(*******************************************************************)
(* Trigger  *)
(*******************************************************************)
(* Zurücksetzen *)
IF xIN_RESET THEN
    iPreStep  := ST160_CETA_e.RESET;
    iOUT_Step := ST160_CETA_e.RESET;
END_IF;

(* Error Quittieren *)
IF (bOUT_Error <> 0) AND xIN_Quit THEN
    xOUT_ErrFlag := FALSE;
    bOUT_Error   := 0;
    iOUT_Step    := ST160_CETA_e.INIT;
END_IF;

(*******************************************************************)
(* Timer *)
(*******************************************************************)
TON_Timeout(IN := xIN_NextStep AND (iLastStep = iOUT_Step) (*todo FG *) ,
            PT := tIN_Timeout);

(*******************************************************************)
(* Bausteine *)
(*******************************************************************)
fb_PnpVerAxis(config          := axis_01Z_LinearConfig,
              xIN_Init        := enIN_State = enState.StateINIT,
              xIN_Reset       := xIN_Reset,
              lrIN_CurrPos    := fb_axis160_01Z.rOUT_ActPos,
              lrIN_Delta_mm   := 0.05,
              iIN_CurrentStep := iOUT_Step,
              iIN_moveNumber  := ST160_PnpVerPos_e._max);

simu_axis160_01Z(xIN_InSimu    := CETA_SIMULATION AND CONST.USE_SIMULATION,
                 rIN_PosActual := fb_axis160_01Z.rOUT_ActPos,
                 pIN_axisSimu  := ADR(axisRef_Simulation),
                 pIN_axisHW    := ADR(axisRef_Hardware),
                 rIN_PosMax    := constAxis_01Z_Beckhoff.POS_MAX,
                 rIN_PosMin    := constAxis_01Z_Beckhoff.POS_MIN,
                 rIN_PixMax    := 80,
                 rIN_PixMin    := 0);

fb_axis160_01Z(enIN_State       := enIN_State,
               parIN_Buttons    := axis_01Z_parIN_Buttons,
               xIN_DisButtons   :=,
               xIN_Quit         := xIN_Quit,
               xIN_AX5000       := TRUE,
               xIN_ENC_ABS      := TRUE, // TODO set accordingly
               xIN_PARAMok      := TRUE,
               xIN_FREE         := TRUE,
               xIN_FREE_HOME    := TRUE,
               rIN_POSMIN       := constAxis_01Z_Beckhoff.POS_MIN,
               rIN_POSMAX       := constAxis_01Z_Beckhoff.POS_MAX,
               rIN_VELOMAX      := constAxis_01Z_Beckhoff.VELO_MAX,
               rIN_VELOMANU     := constAxis_01Z_Beckhoff.VELO_MANU,
               rIN_VELOOPEN     := constAxis_01Z_Beckhoff.POS_MAX / 4,
               rIN_JogInc       := AXIS.rTeachIncAxis,
               rIN_VeloJogManu  := TO_REAL(AXIS.rJogVelo_pc),
               xIN_HomeExe      :=,
               xIN_HomeCalib    :=,
               xIN_Execute      := fb_PnpVerAxis.xOUT_Execute,
               xIN_HomeExe      :=,
               xIN_Relative     :=,
               rIN_Position     := TO_REAL(fb_PnpVerAxis.OUT_MoveProfile.lrPosition),
               rIN_Velocity     := TO_REAL(fb_PnpVerAxis.OUT_MoveProfile.lrVelocity),
               rIN_Acceleration := TO_REAL(fb_PnpVerAxis.OUT_MoveProfile.lrAccel),
               rIN_Deceleration := TO_REAL(fb_PnpVerAxis.OUT_MoveProfile.lrDecel),
               rIN_Jerk         := TO_REAL(fb_PnpVerAxis.OUT_MoveProfile.lrJerk),
               rIN_PosManu      := TO_REAL(axis_01Z_LinearConfig
                                               .movesList[AXIS.bTeachPos[iSelectedAxis]].lrPosition),
               xIN_Reset := (ST160_CETA_e.RESET = iOUT_Step) OR xIN_Reset,
               // output
               rOUT_ActPos => refAxis_01Z_beckhoff.rActPos,
               axisIN_REF  := simu_axis160_01Z.pOUT_axisRef^);

// pneumatics
fb_capMainteningLeft(xIN_Reset    := xIN_Reset OR (ST160_CETA_e.RESET = iOUT_Step),
                     xIN_Quit     := xIN_Quit,
                     xIN_Manu     := enState.StateMANU = enIN_State,
                     pbtIN_Button := ADR(refCylinderBp[1]),
                     xIN_GS       := simu_capMainteningLeft.xOUT_inGS,
                     xIN_AS       := simu_capMainteningLeft.xOUT_inAS,
                     xIN_FREE     := TRUE,
                     xINtoGS      := (ST160_CETA_e.Init_pneumatics = iOUT_Step) OR
                                     (ST160_CETA_e.handling_up = iOUT_Step),
                     xINtoAS   := IN_recipe.Use_element_left AND (ST160_CETA_e.handling_down = iOUT_Step),
                     tIN_ErrAS := DINT_TO_TIME(refCylinderConf
                                                   [ST160_Cylinders_e.Niederhalter_links].toAS_alarm_time),
                     tIN_ErrGS := DINT_TO_TIME(refCylinderConf
                                                   [ST160_Cylinders_e.Niederhalter_links].toGS_alarm_time),
                     tIN_WaitAS := DINT_TO_TIME(refCylinderConf
                                                    [ST160_Cylinders_e.Niederhalter_links].toAS_wait_time),
                     tIN_WaitGS := DINT_TO_TIME(refCylinderConf
                                                    [ST160_Cylinders_e.Niederhalter_links].toGS_wait_time));

simu_capMainteningLeft(xIN_Enable := TRUE, // CETA_SIMULATION AND CONST.USE_SIMULATION,
                       xIN_inGS   := UINT_TO_INT(uiIN_DisplacementSensorLeft) < 10,
                       xIN_inAS   := UINT_TO_INT(uiIN_DisplacementSensorLeft) > 200,
                       xIN_valve  := fb_capMainteningLeft.xOUT_VALVE,
                       tIN_GS_ms  := 200,  // ms
                       tIN_AS_ms  := 200); // ms

fb_capMainteningRight(xIN_Reset    := xIN_Reset OR (ST160_CETA_e.RESET = iOUT_Step),
                      xIN_Quit     := xIN_Quit,
                      xIN_Manu     := enState.StateMANU = enIN_State,
                      pbtIN_Button := ADR(refCylinderBp[2]),
                      xIN_GS       := simu_capMainteningRight.xOUT_inGS,
                      xIN_AS       := simu_capMainteningRight.xOUT_inAS,
                      xIN_FREE     := TRUE,
                      xINtoGS      := (ST160_CETA_e.Init_pneumatics = iOUT_Step) OR
                                      (ST160_CETA_e.handling_up = iOUT_Step),
                      xINtoAS := IN_recipe.Use_element_right AND (ST160_CETA_e.handling_down = iOUT_Step),
                      tIN_ErrAS
                          := DINT_TO_TIME(refCylinderConf
                                              [ST160_Cylinders_e.Niederhalter_rechts].toAS_alarm_time),
                      tIN_ErrGS := DINT_TO_TIME(refCylinderConf
                                                    [ST160_Cylinders_e.Niederhalter_rechts].toGS_alarm_time),
                      tIN_WaitAS := DINT_TO_TIME(refCylinderConf
                                                     [ST160_Cylinders_e.Niederhalter_rechts].toAS_wait_time),
                      tIN_WaitGS := DINT_TO_TIME(refCylinderConf
                                                     [ST160_Cylinders_e.Niederhalter_rechts].toGS_wait_time));

simu_capMainteningRight(xIN_Enable := TRUE, // CETA_SIMULATION AND CONST.USE_SIMULATION,
                        xIN_inGS   := UINT_TO_INT(uiIN_DisplacementSensorRight) < 10,
                        xIN_inAS   := UINT_TO_INT(uiIN_DisplacementSensorRight) > 200,
                        xIN_valve  := fb_capMainteningRight.xOUT_VALVE,
                        tIN_GS_ms  := 200,  // ms
                        tIN_AS_ms  := 200); // ms

fb_dichtung_left(xIN_Reset    := xIN_Reset OR (ST160_CETA_e.RESET = iOUT_Step),
                 xIN_Quit     := xIN_Quit,
                 xIN_Manu     := enState.StateMANU = enIN_State,
                 pbtIN_Button := ADR(refCylinderBp[3]),
                 xIN_GS       := simu_dichtung_left.xOUT_inGS,
                 xIN_AS       := simu_dichtung_left.xOUT_inAS,
                 xIN_FREE     := TRUE,
                 xINtoGS      := (ST160_CETA_e.Init_pneumatics = iOUT_Step) OR
                                 (ST160_CETA_e.unseal_piece = iOUT_Step),
                 xINtoAS   := IN_recipe.Use_element_left AND (ST160_CETA_e.seal_piece = iOUT_Step),
                 tIN_ErrAS := DINT_TO_TIME(refCylinderConf
                                               [ST160_Cylinders_e.Dichtung_prufglocke_links].toAS_alarm_time),
                 tIN_ErrGS := DINT_TO_TIME(refCylinderConf
                                               [ST160_Cylinders_e.Dichtung_prufglocke_links].toGS_alarm_time),
                 tIN_WaitAS := DINT_TO_TIME(refCylinderConf
                                                [ST160_Cylinders_e.Dichtung_prufglocke_links].toAS_wait_time),
                 tIN_WaitGS := DINT_TO_TIME(refCylinderConf
                                                [ST160_Cylinders_e.Dichtung_prufglocke_links].toGS_wait_time));

simu_dichtung_left(xIN_Enable := TRUE,                             // CETA_SIMULATION AND CONST.USE_SIMULATION,
                   xIN_inGS   := NOT fb_dichtung_right.xOUT_VALVE, // no sensor here
                   xIN_inAS   := fb_dichtung_right.xOUT_VALVE,     // no sensor here
                   xIN_valve  := fb_dichtung_left.xOUT_VALVE,
                   tIN_GS_ms  := 200,  // ms
                   tIN_AS_ms  := 200); // ms

fb_dichtung_right(xIN_Reset    := xIN_Reset OR (ST160_CETA_e.RESET = iOUT_Step),
                  xIN_Quit     := xIN_Quit,
                  xIN_Manu     := enState.StateMANU = enIN_State,
                  pbtIN_Button := ADR(refCylinderBp[4]),
                  xIN_GS       := simu_dichtung_right.xOUT_inGS,
                  xIN_AS       := simu_dichtung_right.xOUT_inAS,
                  xIN_FREE     := TRUE,
                  xINtoGS      := (ST160_CETA_e.Init_pneumatics = iOUT_Step) OR
                                  (ST160_CETA_e.unseal_piece = iOUT_Step),
                  xINtoAS   := IN_recipe.Use_element_right AND (ST160_CETA_e.seal_piece = iOUT_Step),
                  tIN_ErrAS := DINT_TO_TIME(refCylinderConf
                                                [ST160_Cylinders_e.Dichtung_prufglocke_rechts].toAS_alarm_time),
                  tIN_ErrGS := DINT_TO_TIME(refCylinderConf
                                                [ST160_Cylinders_e.Dichtung_prufglocke_rechts].toGS_alarm_time),
                  tIN_WaitAS := DINT_TO_TIME(refCylinderConf
                                                 [ST160_Cylinders_e.Dichtung_prufglocke_rechts].toAS_wait_time),
                  tIN_WaitGS := DINT_TO_TIME(refCylinderConf
                                                 [ST160_Cylinders_e.Dichtung_prufglocke_rechts].toGS_wait_time));

simu_dichtung_right(xIN_Enable := TRUE,                             // CETA_SIMULATION AND CONST.USE_SIMULATION,
                    xIN_inGS   := NOT fb_dichtung_right.xOUT_VALVE, // no sensor here
                    xIN_inAS   := fb_dichtung_right.xOUT_VALVE,     // no sensor here
                    xIN_valve  := fb_dichtung_right.xOUT_VALVE,
                    tIN_GS_ms  := 200,  // ms
                    tIN_AS_ms  := 200); // ms

(*******************************************************************)
(* OUTPUTS *)
(*******************************************************************)
// Error Flag 
xOUT_ErrFlag := (bOUT_Error <> 0) OR (ST160_CETA_e.ERROR = iOUT_Step);
// Baustein befindet sich im Ablauf 
xOUT_Busy := (iOUT_Step > ST160_CETA_e.READY) AND (iOUT_Step < ST160_CETA_e.DONE);
// Baustein hat den Ablauf beendet
xOUT_Done := (iOUT_Step = ST160_CETA_e.DONE);
// Process ready
xOUT_Ready := (iOUT_Step = ST160_CETA_e.READY) OR (iOUT_Step = ST160_CETA_e.waitOnMover);
// Timeout FB 				 		
xOUT_Timeout := TON_Timeout.Q;
// Itialisierung fertig			
xOUT_InitDone := (iOUT_Step = ST160_CETA_e.READY) OR (iOUT_Step = ST160_CETA_e.waitOnMover);
// Aktueller Schritt			
iOUT_Step := iOUT_Step; //Im Ablauf gesetzt		
sOUT_Step := TO_STRING(iOUT_Step);
//Fehlernummer	 
bOUT_Error := bOUT_Error; //Im Ablauf/FB gesetzt	
(* Warte (alle Schritte wo auf FG oder Teile gewartet wird) *)
xOUT_Wait := (iOUT_Step = ST160_CETA_e.DONE) OR
             (iOUT_Step = ST160_CETA_e.READY) OR
             (iOUT_Step = ST160_CETA_e.START) OR
             (iOUT_Step = ST160_CETA_e.waitOnMover) OR
             (iOUT_Step = ST160_CETA_e.SYNC_MOVER_LEAVE);

xOUT_MoverFree :=
    NOT (iOUT_Step >= ST160_CETA_e.MOVER_NEEDED_OP AND iOUT_Step < ST160_CETA_e.MOVER_FREE_OP) AND
    (iOUT_Step >= ST160_CETA_e.READY) AND
    (iOUT_Step < ST160_CETA_e.ERROR);

iOUT_ProcessCompletion := F_GetPercent_2(iAktStep,
                                         iAktStep,
                                         iAktStep,
                                         ST160_CETA_e.Init_pneumatics,
                                         ST160_CETA_e.SYNC_MOVER_LEAVE);

xOUT_niederhalter_links :=
    fb_capMainteningLeft.xOUT_VALVE AND NOT (CETA_SIMULATION AND CONST.USE_SIMULATION);

xOUT_niederhalter_rechts :=
    fb_capMainteningRight.xOUT_VALVE AND NOT (CETA_SIMULATION AND CONST.USE_SIMULATION);

xOUT_dichtung_pruflocker_links :=
    fb_dichtung_left.xOUT_VALVE AND NOT (CETA_SIMULATION AND CONST.USE_SIMULATION);

xOUT_dichtung_pruflocker_rechts :=
    fb_dichtung_right.xOUT_VALVE AND NOT (CETA_SIMULATION AND CONST.USE_SIMULATION);

(*******************************************************************)
(* Ablauf *)
(*******************************************************************)

(* Sperren *)
IF xIN_Sperre THEN
    iPreStep  := ST160_CETA_e.RESET;
    iOUT_Step := ST160_CETA_e.RESET;
    RETURN;
END_IF;

(* Schritt Merker *)
IF iAktStep <> iOUT_Step THEN
    iLastStep := iAktStep;
    iAktStep  := iOUT_Step;
END_IF

(* START *)
rtSTART(CLK := xIN_Start);

IF 0 = bOUT_Error THEN
    IF fb_axis160_01Z.xOUT_ErrFlag THEN
        bOUT_Error := 11;
    ELSIF fb_capMainteningLeft.xOUT_ErrFlag THEN
        bOUT_Error := 12;
    ELSIF fb_capMainteningRight.xOUT_ErrFlag THEN
        bOUT_Error := 13;
    END_IF
ELSIF iOUT_Step < ST160_CETA_e.ERROR THEN
    iOUT_Step := ST160_CETA_e.ERROR;
END_IF

(*******************************************************************)
(* Schrittkette  *)
(*******************************************************************)
CASE iOUT_Step OF

(***** RESET *****)
ST160_CETA_e.RESET: (* Schritt 0-99 *)
    //Initialisierungen
    //Start Init Ablauf
    IF xIN_Init THEN
        iOUT_Step := ST160_CETA_e.INIT;
        //Start Manu Ablauf
    ELSIF enIN_State = StateMANU AND xIN_NextStep THEN
        iOUT_Step := ST160_CETA_e.INIT;
    END_IF;

(***** INIT *****)
ST160_CETA_e.INIT: (* Grundstellung ? *)
    iOUT_Step := ST160_CETA_e.Init_pneumatics;

ST160_CETA_e.Init_pneumatics:
    IF (fb_capMainteningLeft.xOUT_inGS AND fb_capMainteningRight.xOUT_inGS) AND
       (fb_dichtung_left.xOUT_inGS AND fb_dichtung_right.xOUT_inGS) THEN
        iOUT_Step := ST160_CETA_e.Init_vertical_down;
    END_IF

ST160_CETA_e.Init_vertical_down:
    IF fb_PnpVerAxis.MoveTo(ST160_PnpVerPos_e.gs_down).xOUT_InPos THEN
        iOUT_Step := ST160_CETA_e.Init_set_program_number;
    END_IF

ST160_CETA_e.Init_set_program_number:
    IF ref_fb_CETA.SetProgramNumber(IN_recipe.Program_number) THEN
        iOUT_Step := ST160_CETA_e.READY;
    END_IF

(***** READY / INIT DONE *****)
ST160_CETA_e.READY:   (* Start AUTO,END,LEER,STEP *)
    IF xIN_Start THEN //IF rtSTART.Q THEN
        iOUT_Step := ST160_CETA_e.START;
    END_IF

(***** START  ZYKLISCH *****)
ST160_CETA_e.START: (*  *)
    IF xIN_NextStep AND pxFG_Freigabe^ THEN
        iOUT_Step       := ST160_CETA_e.waitOnMover;
        xCETA_Result_OK := FALSE;
    END_IF;

ST160_CETA_e.waitOnMover: (*  *)
    IF xIN_NextStep AND __ISVALIDREF(Mover) THEN
        IF (Mover.GetLastStationDone() >= iIN_StationNumber) OR Mover.IsPieceBad() THEN
            iOUT_Step := ST160_CETA_e.SYNC_MOVER_LEAVE;
        ELSIF Mover.GetLastStationDone() < INT#150 THEN
            iOUT_Step := ST160_CETA_e.SYNC_MOVER_LEAVE;
        ELSE
            iOUT_Step := ST160_CETA_e.handling_down;
        END_IF
    END_IF;

ST160_CETA_e.handling_down:
    IF (NOT IN_recipe.Use_element_left OR fb_capMainteningLeft.xOUT_inAS) AND
       (NOT IN_recipe.Use_element_right OR fb_capMainteningRight.xOUT_inAS) THEN
        iOUT_Step := ST160_CETA_e.vertical_up;
    END_IF

ST160_CETA_e.vertical_up:
    IF fb_PnpVerAxis.MoveTo(ST160_PnpVerPos_e.as_up).xOUT_InPos THEN
        iOUT_Step := ST160_CETA_e.seal_piece;
    END_IF

ST160_CETA_e.seal_piece:
    IF (NOT IN_recipe.Use_element_left OR fb_dichtung_left.xOUT_inAS) AND
       (NOT IN_recipe.Use_element_right OR fb_dichtung_right.xOUT_inAS) THEN
        IF CETA_SIMULATION AND CONST.USE_SIMULATION THEN
            iOUT_Step       := ST160_CETA_e.unseal_piece;
            xCETA_Result_OK := TRUE;
        ELSE
            iOUT_Step := ST160_CETA_e.CETA_start;
        END_IF
    END_IF

ST160_CETA_e.CETA_start:
    IF ref_fb_CETA.xOUT_ReadyToStart THEN
        IF ref_fb_CETA.StartMeasurement() THEN
            iOUT_Step := ST160_CETA_e.CETA_wait_on_result;
        ELSE
            bOUT_Error := 21;
        END_IF
    END_IF

ST160_CETA_e.CETA_wait_on_result:
    IF ref_fb_CETA.xOUT_DataReady THEN
        // this void call is needed to tell CETA function block
        // that we have read the result
        ref_fb_CETA.GetResult();
        xCETA_Result_OK := ref_fb_CETA.xOUT_MeasureOK;
        iOUT_Step       := ST160_CETA_e.unseal_piece;
    END_IF

ST160_CETA_e.unseal_piece:
    IF (NOT IN_recipe.Use_element_left OR fb_dichtung_left.xOUT_inGS) AND
       (NOT IN_recipe.Use_element_right OR fb_dichtung_right.xOUT_inGS) THEN
        iOUT_Step := ST160_CETA_e.vertical_down;
    END_IF

ST160_CETA_e.vertical_down:
    IF fb_PnpVerAxis.MoveTo(ST160_PnpVerPos_e.gs_down).xOUT_InPos THEN
        iOUT_Step := ST160_CETA_e.handling_up;
    END_IF

ST160_CETA_e.handling_up:
    IF fb_capMainteningLeft.xOUT_inGS AND fb_capMainteningRight.xOUT_inGS THEN
        iOUT_Step := ST160_CETA_e.SYNC_MOVER_LEAVE;

        IF __ISVALIDREF(Mover) AND NOT xCETA_Result_OK THEN
            Mover.SetErrorCode(CONCAT(INT_TO_STRING(iIN_StationNumber), '-C'));
            // bOUT_Error := 8; // TODO Remove
            iPreStep   := ST160_CETA_e.SYNC_MOVER_LEAVE;

            IF NOT Mover.SetLastStation(-iIN_StationNumber) THEN
                ASSERT(0);
            END_IF
        ELSIF __ISVALIDREF(Mover) AND xCETA_Result_OK THEN
            IF NOT Mover.SetLastStation(iIN_StationNumber) THEN
                ASSERT(0);
            END_IF
        END_IF
    END_IF

ST160_CETA_e.SYNC_MOVER_LEAVE:
    // The mover needs to be taken by MoverMan
    IF NOT __ISVALIDREF(Mover) THEN
        iOUT_Step := ST160_CETA_e.DONE;
    END_IF

(***** DONE *****)
ST160_CETA_e.DONE: (* Letzter Schritt  *)
    IF NOT xIN_AlarmAktiv THEN
        //AUTO
        IF (enIN_State = StateAUTO) AND xIN_RestartCYCL THEN
            iOUT_Step := ST160_CETA_e.START;
            //STEP / END / LEERFAHREN restart
        ELSIF (enIN_State < StateAUTO) AND (enIN_State >= enState.StateSTEP) AND xIN_RestartCYCL THEN
            iOUT_Step := ST160_CETA_e.START;
            //STEP / END / LEERFAHREN fertig
        ELSIF (enIN_State = StateREADY) THEN
            iOUT_Step := ST160_CETA_e.READY;
        END_IF;
    END_IF;

(************ ERROR *************)
ST160_CETA_e.ERROR: (* ERROR *) ;

END_CASE;

END_FUNCTION_BLOCK

// ---- POUs/20_AUTO/ST16x/CETA/FB_CETA_715.TcPOU
// Manage CETATEST void test
// Use the method to perform actions
// Please call each method only once (Use the command only during transition between step) 
FUNCTION_BLOCK PUBLIC FB_CETA_715
VAR_INPUT
    xIN_StatusBits : CETA_IN_u;            // connect this to the 2 first byte of the input of the CETATEST
    xIN_Data       : ARRAY[0..61] OF BYTE; // connect those 62 bytes right after xIN_StatusBits
    xIN_Reset      : BOOL;                 // Reset errors
END_VAR
VAR_OUTPUT
    xOUT_CommandBits    : CETA_OUT_u;           // connect this to the 2 first byte of the Output of the CETATEST
    xOUT_Data           : ARRAY[0..29] OF BYTE; // connect those 30 bytes right after xIN_StatusBits
    xOUT_DataReady      : BOOL;
    xOUT_Error_Flag     : BOOL;
    bOUT_ErrorCode      : BYTE;
    sOUT_ErrorMessage   : STRING;
    xOUT_Measure_1_GOOD : BOOL; // TRUE when the last measurement in canal 1 was GOOD
    bOUT_Error_1        : BYTE;
    xOUT_Measure_2_GOOD : BOOL; // TRUE when the last measurement in canal 2 was GOOD
    bOUT_Error_2        : BYTE;
    xOUT_ReadyToStart   : BOOL; // you can send a start signal
END_VAR
VAR
    iStep       : INT := 0;
    ton_TimeOut : TON;

    iBlockNumber : INT := 0;

    error_message : CETA_error_handling_t;

    ceta_measurement_data : CETA_Measurement_t;

    xResultGood : BOOL := FALSE;

END_VAR
VAR CONSTANT
    DEFAULT_COMMAND_BIT : UINT := 16#00;
END_VAR


ton_TimeOut(IN := 200 = iStep OR 1100 = iStep, PT := T#10S);

CASE iStep OF

0: // reset
    xOUT_CommandBits.raw := 0;

    IF xIN_StatusBits.bits.b09_communication_possible THEN
        iStep := 100;
    END_IF

100: // ready to take command
    // wait on command and read error when there is one
    IF xIN_StatusBits.bits.b08_error_bit THEN
        iStep       := 1000;
        xResultGood := FALSE;
    END_IF

200: // command is sending, wait on a answer

    IF ton_TimeOut.Q THEN
        iStep             := 1500;
        bOUT_ErrorCode    := 0;
        sOUT_ErrorMessage := 'Command timeout';

    ELSIF xOUT_CommandBits.bits.b00_start_stop THEN
        IF xIN_StatusBits.bits.b00_measurement_complete THEN
            iStep               := 240;
            iBlockNumber        := 0;
            xOUT_Measure_1_GOOD := FALSE;
            xOUT_Measure_2_GOOD := FALSE;
        END_IF

    ELSIF xOUT_CommandBits.bits.b01_send_parameters THEN
        IF xIN_StatusBits.bits.b02_parameters_available THEN
            iStep := 300;
        END_IF

    ELSIF xOUT_CommandBits.bits.b02_request_parameters THEN
        IF xIN_StatusBits.bits.b02_parameters_available THEN
            iStep := 300;
        END_IF

    ELSIF xOUT_CommandBits.bits.b03_request_error_code THEN
        IF xIN_StatusBits.bits.b03_error_code_available THEN
            iStep := 1200;
        END_IF

    ELSIF xOUT_CommandBits.bits.b04_change_front_panel_lock_state THEN
        IF xIN_StatusBits.bits.b04_front_panel_lock_state THEN // TODO
            iStep := 0;
        END_IF

    ELSIF xOUT_CommandBits.bits.b05_assign_program_number THEN
        IF xIN_StatusBits.bits.b05_program_number_assigned THEN
            iStep := 0;
        END_IF

    ELSIF xOUT_CommandBits.bits.b06_request_system_information THEN
        IF xIN_StatusBits.bits.b06_system_information_available THEN
            iStep := 300;
        END_IF

    ELSIF xOUT_CommandBits.bits.b07_request_cycle_counter THEN
        IF xIN_StatusBits.bits.b07_cycle_counter_available THEN
            iStep := 300;
        END_IF

        // ELSIF xOUT_CommandBits.bits.request_next_result_block THEN
        //     IF xIN_StatusBits.bits.ne THEN
        //         iStep := 300;
        //     END_IF
    END_IF

240:

    iStep := 250;

    // copy 
    CASE iBlockNumber OF
    0:
        MEMCPY(ADR(ceta_measurement_data.Block0), ADR(xIN_Data), SIZEOF(ceta_measurement_data.Block0));
    1:
        MEMCPY(ADR(ceta_measurement_data.Block1), ADR(xIN_Data), SIZEOF(ceta_measurement_data.Block1));
    2:
        MEMCPY(ADR(ceta_measurement_data.Block2), ADR(xIN_Data), SIZEOF(ceta_measurement_data.Block2));

    ELSE
        iStep := 1500; // should not read more than 3 blocks !
    END_CASE

    iBlockNumber := iBlockNumber + 1;

250:

    // Here we test for iBlockNumber 1 but we have increment the value before
    IF 2 = iBlockNumber THEN
        xOUT_Measure_1_GOOD := ceta_measurement_data.Block1.Result_chanel_1 = CETA_REsult_e.OK;
        xOUT_Measure_2_GOOD := ceta_measurement_data.Block1.Result_chanel_2 = CETA_REsult_e.OK;

        IF NOT xOUT_Measure_1_GOOD THEN
            bOUT_Error_1 := ceta_measurement_data.Block1.Result_chanel_1;
        ELSE
            bOUT_Error_1 := 0;
        END_IF

        IF NOT xOUT_Measure_2_GOOD THEN
            bOUT_Error_2 := ceta_measurement_data.Block1.Result_chanel_2;
        ELSE
            bOUT_Error_2 := 0;
        END_IF
    END_IF

    IF xIN_StatusBits.bits.b11_result_block_handshake_bit THEN
        iStep := 260;
    ELSE
        iStep := 300;
    END_IF

260:
    IF NOT xIN_StatusBits.bits.b11_result_block_handshake_bit THEN
        iStep := 240;
    END_IF

    xOUT_CommandBits.bits.b11_request_next_result_block := xIN_StatusBits.bits.b11_result_block_handshake_bit;

300: // data available
    xOUT_CommandBits.raw := 0;
// Use the read() method to return to state 100

1000: // read error code
    xOUT_CommandBits.raw := 0;
    //
    xOUT_CommandBits.bits.b03_request_error_code := TRUE;

    iStep := 1100;

1100: // read error code
    IF ton_TimeOut.Q THEN
        iStep := 0; // reset .. there is nothing we can do
    ELSIF xIN_StatusBits.bits.b03_error_code_available THEN
        iStep := 1200;
    END_IF

1200: // read error
    error_message.command_in_error.raw := xIN_Data[0] + SHL(TO_UINT(xIN_Data[1]), 8);

    bOUT_ErrorCode := error_message.error_code;

    IF 0 = error_message.command_in_error.raw THEN
        sOUT_ErrorMessage := 'CETA in error, not due to Ethercat communication';

    ELSIF xOUT_CommandBits.bits.b01_send_parameters THEN
        sOUT_ErrorMessage := 'send_parameters command failed';

    ELSIF xOUT_CommandBits.bits.b02_request_parameters THEN
        sOUT_ErrorMessage := 'request_parameters command failed';

    ELSIF xOUT_CommandBits.bits.b03_request_error_code THEN
        sOUT_ErrorMessage := 'request_error_code command failed';

    ELSIF xOUT_CommandBits.bits.b04_change_front_panel_lock_state THEN
        sOUT_ErrorMessage := 'change_front_panel_lock_state command failed';

    ELSIF xOUT_CommandBits.bits.b05_assign_program_number THEN
        sOUT_ErrorMessage := 'assign_program_number command failed';

    ELSIF xOUT_CommandBits.bits.b06_request_system_information THEN
        sOUT_ErrorMessage := 'request_system_information command failed';

    ELSIF xOUT_CommandBits.bits.b07_request_cycle_counter THEN
        sOUT_ErrorMessage := 'request_cycle_counter command failed';

    END_IF

    iStep := 1500;

1500: // in error, wait on reset
    IF xIN_Reset THEN
        sOUT_ErrorMessage                         := '';
        bOUT_ErrorCode                            := 0;
        xOUT_CommandBits.raw                      := 0;
        xOUT_CommandBits.bits.b08_reset_error_bit := TRUE;
        iStep                                     := 0;
    END_IF

END_CASE

xOUT_DataReady    := 300 = iStep;
xOUT_Error_Flag   := 1500 = iStep;
xOUT_ReadyToStart := xIN_StatusBits.bits.b10_device_ready_to_start;

METHOD GetParameter : BOOL
VAR_INPUT
END_VAR
END_METHOD

METHOD GetResult : BOOL
VAR_INPUT
END_VAR
IF 300 = THIS^.iStep THEN
    GetResult   := TRUE;
    THIS^.iStep := 0;
ELSE
    GetResult := FALSE;
END_IF
END_METHOD

METHOD SetProgramNumber : BOOL
VAR_INPUT
	program_number : USINT;
END_VAR
IF 100 = THIS^.iStep THEN
	THIS^.iStep := 200;
	THIS^.xOUT_CommandBits.bits.b05_assign_program_number := TRUE;
	THIS^.xOUT_Data[0] := USINT_TO_BYTE(program_number);
	SetProgramNumber := TRUE;
ELSE
    THIS^.iStep      := 0;
	SetProgramNumber := FALSE;
END_IF
END_METHOD

METHOD StartMeasurement : BOOL
VAR_INPUT
END_VAR
IF 100 = THIS^.iStep THEN
    THIS^.iStep                                := 200;
    THIS^.xOUT_CommandBits.bits.b00_start_stop := TRUE;
    StartMeasurement                           := TRUE;
ELSE
    THIS^.iStep      := 0;
    StartMeasurement := FALSE;
END_IF
END_METHOD

END_FUNCTION_BLOCK

// ---- POUs/20_AUTO/ST16x/FB_AUT_165.TcPOU
FUNCTION_BLOCK FB_AUT_165 EXTENDS FB_AUT_ABSTRACT
(****************************************************************************)
(*	POU_AUT_zxx			Bausteinaufrufe Station	zxx							*)
(*	Status				ungetestet											*)
(*  Version:			1.0													*)
(*	Beschrieb:																*)
(*																			*)
(*	Abläufe:			FB_ABLzxxA		Hauptablauf							*)
(*																			*)
(*																			*)
(* 	25.09.2019/Dj															*)
(****************************************************************************)
(*	dd.mm.yyyy   KZ    x.y			Beschrieb								*)
(****************************************************************************)
VAR_INPUT
    (* spezifische Eingänge *)

END_VAR
VAR_OUTPUT
    (* spezifische Ausgänge *)

END_VAR
VAR
    (* Bausteine *)
    fb_ABL_CETA : FB_ABL_160;
	
	fb_CETA : FB_CETA_715;

    fb_stat : FB_AUT_Statistics;

END_VAR

(*******************************************************************)
(* Timer *)
(*******************************************************************)

(*******************************************************************)
(* Flanken / Merker *)
(*******************************************************************)
//MANU CYCLE
IF (enIN_State = StateMANU) AND xIN_ManuCycle THEN
    xManuCycle := TRUE;
END_IF;

IF (enIN_State <> StateMANU) OR xOUT_Done THEN
    xManuCycle := FALSE;
END_IF

//NEXT STEP
xNextStep := (enIN_State > StateSTEP) OR
             ((enIN_State = StateSTEP) AND xIN_Step) OR
             ((enIN_State = StateMANU) AND xManuCycle);

//RESET
xReset := (enIN_State < StateREADY) AND (enIN_State <> StateINIT) AND NOT xManuCycle;

(*******************************************************************)
(* Bausteinaufrufe Abläufe *)
(*******************************************************************)

xRelease := MAIN.MoverMan.IsProcessUsed(THIS^);

fb_CETA(xIN_StatusBits   := CETA_IO.I_ST165_StatusBits,
        xIN_Data         := CETA_IO.I_ST165_Data,
        xIN_Reset        := xReset OR xIN_Quit,
        xOUT_CommandBits => CETA_IO.Q_ST165_CommandBits,
        xOUT_Data        => CETA_IO.Q_ST165_Data);

fb_ABL_CETA(xIN_Reset       := xReset,
            xIN_Init        := xIN_Init,
            xIN_Quit        := xIN_Quit,
            xIN_Start       := enIN_State >= enState.StateLEER AND xRelease,
            xIN_Sperre      := NOT xIN_On,
            xIN_NextStep    := xNextStep,
            xIN_AlarmAktiv  := xIN_AlarmAktiv,
            xIN_DryCycle    := xIN_DryCycle,
            xIN_RestartCYCL := enIN_State >= enState.StateLEER,
            enIN_State      := enIN_State,
            tIN_Timeout     := tIN_Timeout,
            pxFG_Freigabe   := ADR(xRelease),
            // CleverTrackLib
            Mover := THIS^.Mover,
            // for multiple reference of the FB
            ref_fb_CETA := fb_CETA,

            refAxis_01Z_beckhoff         := ST16x_Axis.axis165_01Z,
            constAxis_01Z_Beckhoff       := ST16x_Axis.const165_01Z,
            axis_01Z_LinearConfig        := _20_AUTO.recipe.linearAxis[LinearAxis_e.ST165_01Z],
            iSelectedAxis                := Axis_e.ST165_01Z,
            axis_01Z_parIN_Buttons       := ADR(AXIS.btTeachArAxis[Axis_e.ST165_01Z]),
            refCylinderBp                := HMI.btManuCylinders[StationList_e.ST165],
            refCylinderConf              := _20_AUTO.recipe.cylinder2Pos[StationList_e.ST165],
            uiIN_DisplacementSensorLeft  := IO_BOX.I3200_ST165_Wegmessenor_links,
            uiIN_DisplacementSensorRight := IO_BOX.I3300_ST165_Wegmessenor_rechts,
            IN_recipe                    := _20_AUTO.recipe.st165,
            iIN_StationNumber            := 165,

            xOUT_niederhalter_links         => IO_BOX.Q0304_14_ST165_niederhalter_links,
            xOUT_niederhalter_rechts        => IO_BOX.Q0305_14_ST165_niederhalter_rechts,
            xOUT_dichtung_pruflocker_links  => IO_BOX.Q0306_14_ST165_dichtung_pruflocker_links,
            xOUT_dichtung_pruflocker_rechts => IO_BOX.Q0306_12_ST165_dichtung_pruflocker_rechts,

            axisRef_Hardware   := ST16x_Axis.axis165_01Z.axis,
            axisRef_Simulation := SIMU.axis_ref[Axis_e.ST165_01Z]);
			
fb_stat(xIN_Enable  := enState.StateAUTO = enIN_State,
        xIN_Waiting := fb_ABL_CETA.xOUT_Wait,
        xIN_Running := (fb_ABL_CETA.iOUT_Step >= ST160_CETA_e.START) AND
                       (fb_ABL_CETA.iOUT_Step <= ST160_CETA_e.DONE),
        // Since we use a mover system, a cycle is done when we are waiting on a mover
        xIN_Done := fb_ABL_CETA.iOUT_Step = ST160_CETA_e.waitOnMover);

(*******************************************************************)
(* Mover reset flags *)
(*******************************************************************)

(*******************************************************************)
(* OUTPUT *)
(*******************************************************************)
xOUT_InitDone := fb_ABL_CETA.xOUT_InitDone;
xOUT_Ready    := fb_ABL_CETA.xOUT_Ready;
xOUT_Done     := fb_ABL_CETA.xOUT_Done;
xOUT_ErrFlag  := fb_ABL_CETA.xOUT_ErrFlag;
xOUT_Wait     := fb_ABL_CETA.xOUT_Wait;
xOUT_AlarmST  := xOUT_ErrFlag;

(*******************************************************************)
(* Bausteinaufruf Error Station *)
(*******************************************************************)
// POU_ERR_VORLAGE(xIN_QUIT:=xIN_Quit , pstrArIN_ALARM:=ADR(HMI.strArALARM[1]));

(* % of completion of the process *)
PROPERTY iCompletionPC : INT
GET
iCompletionPC := THIS^.fb_ABL_CETA.iOUT_ProcessCompletion;
END_GET
END_PROPERTY

PROPERTY ProcessExecution : ProcessExecution_e
GET
ProcessExecution := THIS^._ProcessExecution;
END_GET
SET
THIS^._ProcessExecution := ProcessExecution;
END_SET
END_PROPERTY

PROPERTY xBusy : BOOL
GET
xBusy := THIS^.fb_ABL_CETA.xOUT_Busy;
END_GET
SET
END_SET
END_PROPERTY

PROPERTY xDone : BOOL
GET
xDone := THIS^.fb_ABL_CETA.xOUT_Ready OR THIS^.fb_ABL_CETA.xOUT_Done;
END_GET
END_PROPERTY

PROPERTY xMoverPathFree : BOOL
GET
xMoverPathFree := THIS^.fb_ABL_CETA.xOUT_MoverFree OR THIS^.fb_ABL_CETA.xOUT_Ready OR THIS^.fb_ABL_CETA.xOUT_Done;
END_GET
END_PROPERTY

PROPERTY xMoverShouldLeave : BOOL
GET
xMoverShouldLeave := THIS^.fb_ABL_CETA.iOUT_Step = ST160_CETA_e.SYNC_MOVER_LEAVE;
END_GET
END_PROPERTY

END_FUNCTION_BLOCK

// ---- POUs/20_AUTO/ST170/FB_AUT_170.TcPOU
FUNCTION_BLOCK FB_AUT_170 EXTENDS FB_AUT_ABSTRACT
(****************************************************************************)
(*	POU_AUT_zxx			Bausteinaufrufe Station	zxx							*)
(*	Status				ungetestet											*)
(*  Version:			1.0													*)
(*	Beschrieb:																*)
(*																			*)
(*	Abläufe:			FB_ABLzxxA		Hauptablauf							*)
(*																			*)
(*																			*)
(* 	25.09.2019/Dj															*)
(****************************************************************************)
(*	dd.mm.yyyy   KZ    x.y			Beschrieb								*)
(****************************************************************************)
VAR_INPUT
    (* spezifische Eingänge *)

END_VAR
VAR_OUTPUT
    (* spezifische Ausgänge *)

END_VAR
VAR
    (* Bausteine *)
    fb_ABL_RFID : FB_ABL_170;

    fb_stat : FB_AUT_Statistics;

END_VAR

(*******************************************************************)
(* Timer *)
(*******************************************************************)

(*******************************************************************)
(* Flanken / Merker *)
(*******************************************************************)
//MANU CYCLE
IF (enIN_State = StateMANU) AND xIN_ManuCycle THEN
    xManuCycle := TRUE;
END_IF;

IF (enIN_State <> StateMANU) OR xOUT_Done THEN
    xManuCycle := FALSE;
END_IF

//NEXT STEP
xNextStep := (enIN_State > StateSTEP) OR
             ((enIN_State = StateSTEP) AND xIN_Step) OR
             ((enIN_State = StateMANU) AND xManuCycle);

//RESET
xReset := (enIN_State < StateREADY) AND (enIN_State <> StateINIT) AND NOT xManuCycle;

(*******************************************************************)
(* Bausteinaufrufe Abläufe *)
(*******************************************************************)

xRelease := MAIN.MoverMan.IsProcessUsed(THIS^);

fb_ABL_RFID(xIN_Reset       := xReset,
            xIN_Init        := xIN_Init,
            xIN_Quit        := xIN_Quit,
            xIN_Start       := enIN_State >= enState.StateLEER AND xRelease,
            xIN_Sperre      := NOT xIN_On,
            xIN_NextStep    := xNextStep,
            xIN_AlarmAktiv  := xIN_AlarmAktiv,
            xIN_DryCycle    := xIN_DryCycle,
            xIN_RestartCYCL := enIN_State >= enState.StateLEER,
            enIN_State      := enIN_State,
            tIN_Timeout     := tIN_Timeout,
            pxFG_Freigabe   := ADR(xRelease),
            // CleverTrackLib
            Mover := THIS^.Mover);

fb_stat(xIN_Enable  := enState.StateAUTO = enIN_State,
        xIN_Waiting := fb_ABL_RFID.xOUT_Wait,
        xIN_Running := (fb_ABL_RFID.iOUT_Step >= ST170_RFID_e.START) AND
                       (fb_ABL_RFID.iOUT_Step <= ST170_RFID_e.DONE),
        // Since we use a mover system, a cycle is done when we are waiting on a mover
        xIN_Done := fb_ABL_RFID.iOUT_Step = ST170_RFID_e.waitOnMover);

(*******************************************************************)
(* Mover reset flags *)
(*******************************************************************)

(*******************************************************************)
(* OUTPUT *)
(*******************************************************************)
xOUT_InitDone := fb_ABL_RFID.xOUT_InitDone;
xOUT_Ready    := fb_ABL_RFID.xOUT_Ready;
xOUT_Done     := fb_ABL_RFID.xOUT_Done;
xOUT_ErrFlag  := fb_ABL_RFID.xOUT_ErrFlag;
xOUT_Wait     := fb_ABL_RFID.xOUT_Wait;
xOUT_AlarmST  := xOUT_ErrFlag;

(*******************************************************************)
(* Bausteinaufruf Error Station *)
(*******************************************************************)
// POU_ERR_VORLAGE(xIN_QUIT:=xIN_Quit , pstrArIN_ALARM:=ADR(HMI.strArALARM[1]));

(* % of completion of the process *)
PROPERTY iCompletionPC : INT
GET
iCompletionPC := THIS^.fb_ABL_RFID.iOUT_ProcessCompletion;
END_GET
END_PROPERTY

PROPERTY ProcessExecution : ProcessExecution_e
GET
ProcessExecution := THIS^._ProcessExecution;
END_GET
SET
THIS^._ProcessExecution := ProcessExecution;
END_SET
END_PROPERTY

PROPERTY xBusy : BOOL
GET
xBusy := THIS^.fb_ABL_RFID.xOUT_Busy;
END_GET
SET
END_SET
END_PROPERTY

PROPERTY xDone : BOOL
GET
xDone := THIS^.fb_ABL_RFID.xOUT_Ready OR THIS^.fb_ABL_RFID.xOUT_Done;
END_GET
END_PROPERTY

PROPERTY xMoverPathFree : BOOL
GET
xMoverPathFree := THIS^.fb_ABL_RFID.xOUT_MoverFree OR THIS^.fb_ABL_RFID.xOUT_Ready OR THIS^.fb_ABL_RFID.xOUT_Done;
END_GET
END_PROPERTY

PROPERTY xMoverShouldLeave : BOOL
GET
xMoverShouldLeave := THIS^.fb_ABL_RFID.iOUT_Step = ST170_RFID_e.SYNC_MOVER_LEAVE;
END_GET
END_PROPERTY

END_FUNCTION_BLOCK

// ---- POUs/20_AUTO/ST170/FB_ABL_170.TcPOU
FUNCTION_BLOCK FB_ABL_170
(****************************************************************************************)
(*	TITEL				laden kristall- Modul	    										*)
(*	Status				ungetestet                         								*)
(*	Beschrieb:			Ablaufbeschreibung												*)
(*																						*)
(*	Steps:	self-explained using enum													*)
(***********************************Revisionen*******************************************)
(*	see github blames																	*)
(****************************************************************************************)

VAR_INPUT
    xIN_Reset       : BOOL;          // Schrittkette zurücksetzen 
    xIN_Init        : BOOL;          // Initialisieren
    xIN_Quit        : BOOL;          // Fehler quittieren 
    xIN_Start       : BOOL;          // Startbefehl
    xIN_Sperre      : BOOL;          // FB Sperren 
    xIN_NextStep    : BOOL;          // Nächsten Schritt ausführen 
    xIN_AlarmAktiv  : BOOL;          // Anlage hat Alarm
    xIN_DryCycle    : BOOL;          // Fahren ohne Teile
    xIN_RestartCYCL : BOOL;          // Zyklus erneut starten im STEP, END, LEERFAHREN
    enIN_State      : enState;       // Status Anlage
    tIN_Timeout     : TIME := T#10s; // Timout

    pxFG_Freigabe : POINTER TO BOOL; //Freigabe von Station

    // Application specific
    Mover : REFERENCE TO FB_Mover;

END_VAR
VAR_OUTPUT
    (* standart Ausgänge *)
    xOUT_ErrFlag  : BOOL;         // Error Flag 
    xOUT_Busy     : BOOL;         // Baustein befindet sich im Ablauf 
    xOUT_Done     : BOOL;         // Baustein hat den Ablauf beendet 		
    xOUT_Ready    : BOOL;         // Ready to begin, should be the same state as done	
    xOUT_Timeout  : BOOL;         // Timeout FB 
    xOUT_InitDone : BOOL;         // initialisierung fertig
    xOUT_Wait     : BOOL;         // Wartet auf Bedingung
    iOUT_Step     : ST170_RFID_e; // Aktueller Schritt 
    sOUT_Step     : STRING;       // Aktueller Schritt but in string format
    bOUT_Error    : BYTE;         // Fehlernummer

    iOUT_ProcessCompletion : INT;  //process completion, express in % (0-100)
    xOUT_MoverFree         : BOOL; // The mover is free to move
END_VAR
VAR
    (* Standard *)
    (* Schritt *)
    iLastStep : ST170_RFID_e; // Merker letzter Schritt 
    iPreStep  : ST170_RFID_e; // Schritt zurück nach Alarm 
    iAktStep  : ST170_RFID_e; // aktueller Schritt

    // Trigger Starten 
    rtSTART : R_TRIG;
    // Timer TimeOut 
    TON_Timeout : TON;

    (* Bausteine *)
    fb_PnpVerAxis    : FB_LinearMotionMan;
    simu_axis170_01Z : FB_Simu_AxisLM_V1_1;
    fb_axis170_01Z   : FB_AxisLM_V1_1;

    (* Spezial *)
    xRFID_Result_Left_OK  : BOOL;
    xRFID_Result_Right_OK : BOOL;

END_VAR
VAR CONSTANT
    RFID_SIMULATION : BOOL := FALSE; // Set to TRUE to simulate this part of the program
END_VAR

(*******************************************************************)
(* Trigger  *)
(*******************************************************************)
(* Zurücksetzen *)
IF xIN_RESET THEN
    iPreStep  := ST170_RFID_e.RESET;
    iOUT_Step := ST170_RFID_e.RESET;
END_IF;

(* Error Quittieren *)
IF (bOUT_Error <> 0) AND xIN_Quit THEN
    xOUT_ErrFlag := FALSE;
    bOUT_Error   := 0;
    iOUT_Step    := iPreStep;
END_IF;

(*******************************************************************)
(* Timer *)
(*******************************************************************)
TON_Timeout(IN := xIN_NextStep AND (iLastStep = iOUT_Step) (*todo FG *) ,
            PT := tIN_Timeout);

(*******************************************************************)
(* Bausteine *)
(*******************************************************************)
fb_PnpVerAxis(config          := _20_AUTO.recipe.linearAxis[LinearAxis_e.ST170_01Z],
              xIN_Init        := enIN_State = enState.StateINIT,
              xIN_Reset       := xIN_Reset,
              lrIN_CurrPos    := fb_axis170_01Z.rOUT_ActPos,
              lrIN_Delta_mm   := 0.5,
              iIN_CurrentStep := iOUT_Step,
              iIN_moveNumber  := ST170_PnpVerPos_e._max);

simu_axis170_01Z(xIN_Enable          := RFID_SIMULATION AND CONST.USE_SIMULATION,
                 bIN_AxisCntr        := fb_axis170_01Z.bOUT_AxisCntr,
                 wIN_AxisState       := ST170_Axis.axis170_01Z.wState,
                 udiIN_HomingTime_ms := 2000,
                 pIN_axisSimu        := ADR(SIMU.axis_ref[Axis_e.ST170_01Z]),
                 pIN_axisHW          := ADR(ST170_Axis.axis170_01Z.axis),
                 rIN_PosActual       := ST170_Axis.axis170_01Z.rActPos,
                 rIN_PosMax          := ST170_Axis.const170_01Z.POS_MAX,
                 rIN_PosMin          := ST170_Axis.const170_01Z.POS_MIN,
                 rIN_PixMax          := 80,
                 rIN_PixMin          := 0);

fb_axis170_01Z(enIN_State       := enIN_State,
               parIN_Buttons    := ADR(AXIS.btTeachArAxis[Axis_e.ST170_01Z]),
               xIN_DisButtons   :=,
               xIN_Quit         := xIN_Quit,
               xIN_PARAMok      := TRUE,
               xIN_FREE         := TRUE,
               xIN_FREE_HOME    := TRUE,
               rIN_POSMIN       := ST170_Axis.const170_01Z.POS_MIN,
               rIN_POSMAX       := ST170_Axis.const170_01Z.POS_MAX,
               rIN_VELOMAX      := ST170_Axis.const170_01Z.VELO_MAX,
               rIN_VELOMANU     := ST170_Axis.const170_01Z.VELO_MANU,
               rIN_VELOOPEN     := ST170_Axis.const170_01Z.POS_MAX / 4,
               rIN_JogInc       := AXIS.rTeachIncAxis,
               xIN_Execute      := fb_PnpVerAxis.xOUT_Execute,
               xIN_Relative     :=,
               xIN_STOP         :=,
               xIN_OFF          :=,
               rIN_Position     := TO_REAL(fb_PnpVerAxis.OUT_MoveProfile.lrPosition),
               rIN_Velocity     := TO_REAL(fb_PnpVerAxis.OUT_MoveProfile.lrVelocity),
               rIN_Acceleration := TO_REAL(fb_PnpVerAxis.OUT_MoveProfile.lrAccel),
               rIN_Deceleration := TO_REAL(fb_PnpVerAxis.OUT_MoveProfile.lrDecel),
               rIN_Jerk         := TO_REAL(fb_PnpVerAxis.OUT_MoveProfile.lrJerk),
               rIN_PosManu      :=
               TO_REAL(_20_AUTO.recipe
                           .linearAxis[LinearAxis_e.ST170_01Z].movesList[AXIS.bTeachPos[Axis_e.ST170_01Z]].lrPosition),
               rIN_VeloJogManu := TO_REAL(Axis.rJogVelo_pc),
               xIN_Home        := ST170_RFID_e.Init_vertical_homing = iOUT_Step,
               xIN_Reset       := (ST170_RFID_e.RESET = iOUT_Step) OR xIN_Reset,
               wAxisState      := simu_axis170_01Z.wOUT_AxisState,
               bOUT_AxisCntr   => ST170_Axis.axis170_01Z.bCtrlHi,
               rOUT_ActPos     => ST170_Axis.axis170_01Z.rActPos,
               axisIN_REF      := simu_axis170_01Z.pOUT_axisRef^);

(*******************************************************************)
(* OUTPUTS *)
(*******************************************************************)
// Error Flag 
xOUT_ErrFlag := (bOUT_Error <> 0) OR (ST170_RFID_e.ERROR = iOUT_Step);
// Baustein befindet sich im Ablauf 
xOUT_Busy := (iOUT_Step > ST170_RFID_e.READY) AND (iOUT_Step < ST170_RFID_e.DONE);
// Baustein hat den Ablauf beendet
xOUT_Done := (iOUT_Step = ST170_RFID_e.DONE);
// Process ready
xOUT_Ready := (iOUT_Step = ST170_RFID_e.READY) OR (iOUT_Step = ST170_RFID_e.waitOnMover);
// Timeout FB 				 		
xOUT_Timeout := TON_Timeout.Q;
// Itialisierung fertig			
xOUT_InitDone := (iOUT_Step = ST170_RFID_e.READY) OR (iOUT_Step = ST170_RFID_e.waitOnMover);
// Aktueller Schritt			
iOUT_Step := iOUT_Step; //Im Ablauf gesetzt		
sOUT_Step := TO_STRING(iOUT_Step);
//Fehlernummer	 
bOUT_Error := bOUT_Error; //Im Ablauf/FB gesetzt	
(* Warte (alle Schritte wo auf FG oder Teile gewartet wird) *)
xOUT_Wait := (iOUT_Step = ST170_RFID_e.DONE) OR
             (iOUT_Step = ST170_RFID_e.READY) OR
             (iOUT_Step = ST170_RFID_e.START) OR
             (iOUT_Step = ST170_RFID_e.waitOnMover) OR
             (iOUT_Step = ST170_RFID_e.SYNC_MOVER_LEAVE);

xOUT_MoverFree := NOT (iOUT_Step >= ST170_RFID_e.MOVER_NEEDED_OP AND iOUT_Step < ST170_RFID_e.MOVER_FREE_OP) AND
                  (iOUT_Step >= ST170_RFID_e.READY) AND
                  (iOUT_Step < ST170_RFID_e.ERROR);

iOUT_ProcessCompletion := F_GetPercent_2(iAktStep,
                                         iAktStep,
                                         iAktStep,
                                         ST170_RFID_e.vertical_up,
                                         ST170_RFID_e.SYNC_MOVER_LEAVE);

OUT.Q026_ST170_rfid_start_links :=
    _20_AUTO.recipe.st170.Use_element_left AND
    (ST170_RFID_e.RFID_start = iOUT_Step) AND
    NOT xRFID_Result_Left_OK AND // If we redo a flashing, it will generate an error
    NOT (RFID_SIMULATION AND CONST.USE_SIMULATION);

OUT.Q027_ST170_rfid_start_rechts :=
    _20_AUTO.recipe.st170.Use_element_right AND
    (ST170_RFID_e.RFID_start = iOUT_Step) AND
    NOT xRFID_Result_Right_OK AND // If we redo a flashing, it will generate an error
    NOT (RFID_SIMULATION AND CONST.USE_SIMULATION);

OUT.Q040_ST170_RFID_Links_Type_Bit_0  := _20_AUTO.recipe.st170.RFID_Type.0;
OUT.Q041_ST170_RFID_Links_Type_Bit_1  := _20_AUTO.recipe.st170.RFID_Type.1;
OUT.Q042_ST170_RFID_Links_Type_Bit_2  := _20_AUTO.recipe.st170.RFID_Type.2;
OUT.Q043_ST170_RFID_Rechts_Type_Bit_0 := _20_AUTO.recipe.st170.RFID_Type.0;
OUT.Q044_ST170_RFID_Rechts_Type_Bit_1 := _20_AUTO.recipe.st170.RFID_Type.1;
OUT.Q045_ST170_RFID_Rechts_Type_Bit_2 := _20_AUTO.recipe.st170.RFID_Type.2;

(*******************************************************************)
(* Ablauf *)
(*******************************************************************)

(* Sperren *)
IF xIN_Sperre THEN
    iPreStep  := ST170_RFID_e.RESET;
    iOUT_Step := ST170_RFID_e.RESET;
    RETURN;
END_IF;

(* Schritt Merker *)
IF iAktStep <> iOUT_Step THEN
    iLastStep := iAktStep;
    iAktStep  := iOUT_Step;
END_IF

(* START *)
rtSTART(CLK := xIN_Start);

IF 0 = bOUT_Error THEN
    IF fb_axis170_01Z.xOUT_ErrFlag THEN
        bOUT_Error := 11;
    END_IF
ELSIF iOUT_Step < ST170_RFID_e.ERROR THEN
    iOUT_Step := ST170_RFID_e.ERROR;
END_IF

(*******************************************************************)
(* Schrittkette  *)
(*******************************************************************)
CASE iOUT_Step OF

(***** RESET *****)
ST170_RFID_e.RESET: (* Schritt 0-99 *)
    //Initialisierungen
    //Start Init Ablauf
    IF xIN_Init THEN
        iOUT_Step := ST170_RFID_e.INIT;
        //Start Manu Ablauf
    ELSIF enIN_State = StateMANU AND xIN_NextStep THEN
        iOUT_Step := ST170_RFID_e.INIT;
    END_IF;

(***** INIT *****)
ST170_RFID_e.INIT: (* Grundstellung ? *)
    IF fb_axis170_01Z.xOUT_HOMED THEN
        iOUT_Step := ST170_RFID_e.Init_vertical_down;
    ELSE
        iOUT_Step := ST170_RFID_e.Init_vertical_homing;
    END_IF

ST170_RFID_e.Init_vertical_homing:
    IF fb_axis170_01Z.xOUT_HOMED THEN
        iOUT_Step := ST170_RFID_e.Init_vertical_down;
    END_IF

ST170_RFID_e.Init_vertical_down:
    IF fb_PnpVerAxis.MoveTo(ST170_PnpVerPos_e.gs_down).xOUT_InPos THEN
        iOUT_Step := ST170_RFID_e.READY;
    END_IF

(***** READY / INIT DONE *****)
ST170_RFID_e.READY:   (* Start AUTO,END,LEER,STEP *)
    IF xIN_Start THEN //IF rtSTART.Q THEN
        iOUT_Step := ST170_RFID_e.START;
    END_IF

(***** START  ZYKLISCH *****)
ST170_RFID_e.START: (*  *)
    IF xIN_NextStep AND pxFG_Freigabe^ THEN
        iOUT_Step := ST170_RFID_e.waitOnMover;
    END_IF;

ST170_RFID_e.waitOnMover: (*  *)
    IF xIN_NextStep AND __ISVALIDREF(Mover) THEN
        IF (Mover.GetLastStationDone() >= 170) THEN
            iOUT_Step := ST170_RFID_e.SYNC_MOVER_LEAVE;
        ELSIF Mover.GetLastStationDone() < INT#110 THEN
            iOUT_Step := ST170_RFID_e.SYNC_MOVER_LEAVE;
        ELSE
            iOUT_Step := ST170_RFID_e.vertical_up;
        END_IF
    END_IF;

ST170_RFID_e.vertical_up:
    IF xIN_NextStep AND fb_PnpVerAxis.MoveTo(ST170_PnpVerPos_e.as_up).xOUT_InPos THEN
        iOUT_Step             := ST170_RFID_e.RFID_start;
        xRFID_Result_Left_OK  := NOT _20_AUTO.recipe.st170.Use_element_left;  // Force ok result when not used
        xRFID_Result_Right_OK := NOT _20_AUTO.recipe.st170.Use_element_right; // Force ok result when not used
    END_IF

ST170_RFID_e.RFID_start:
    IF xIN_NextStep AND
       (NOT _20_AUTO.recipe.st170.Use_element_left OR NOT IN.I030_rfid_test_link_out1_170_20) AND
       (NOT _20_AUTO.recipe.st170.Use_element_right OR NOT IN.I033_rfid_test_link_out1_170_21) THEN
        iOUT_Step := ST170_RFID_e.RFID_wait_on_result;

        IF __ISVALIDREF(Mover) AND_THEN NOT Mover.SetLastStation(170) THEN
            ASSERT(0);
        END_IF
    END_IF

ST170_RFID_e.RFID_wait_on_result:
    IF xIN_NextStep AND
       (NOT _20_AUTO.recipe.st170.Use_element_left OR IN.I030_rfid_test_link_out1_170_20) AND
       (NOT _20_AUTO.recipe.st170.Use_element_right OR IN.I033_rfid_test_link_out1_170_21) THEN

        xRFID_Result_Left_OK := (NOT _20_AUTO.recipe.st170.Use_element_left OR
                                 (IN.I031_rfid_test_link_out2_170_20 AND NOT IN.I032_rfid_test_link_out3_170_20));

        xRFID_Result_Right_OK := (NOT _20_AUTO.recipe.st170.Use_element_right OR
                                  (IN.I034_rfid_test_link_out2_170_21 AND NOT IN.I035_rfid_test_link_out3_170_21));

        iOUT_Step := ST170_RFID_e.vertical_down;
    END_IF

ST170_RFID_e.vertical_down:
    IF xIN_NextStep AND fb_PnpVerAxis.MoveTo(ST170_PnpVerPos_e.gs_down).xOUT_InPos THEN
        iOUT_Step := ST170_RFID_e.SYNC_MOVER_LEAVE;

        IF __ISVALIDREF(Mover) AND xRFID_Result_Left_OK AND xRFID_Result_Right_OK THEN
            IF NOT Mover.SetLastStation(170) THEN
                ASSERT(0);
            END_IF
        ELSIF __ISVALIDREF(Mover) THEN

            IF NOT xRFID_Result_Left_OK AND NOT xRFID_Result_Right_OK THEN
                Mover.SetErrorCode('170-B Both');

            ELSIF NOT xRFID_Result_Left_OK THEN
                Mover.SetErrorCode('170-B Left');

            ELSIF NOT xRFID_Result_Right_OK THEN
                Mover.SetErrorCode('170-B Right');

            END_IF

            IF NOT Mover.SetLastStation(-170) THEN
                ASSERT(0);
            END_IF
        END_IF
    END_IF

ST170_RFID_e.SYNC_MOVER_LEAVE:
    // The mover needs to be taken by MoverMan
    IF NOT __ISVALIDREF(Mover) THEN
        iOUT_Step := ST170_RFID_e.DONE;
    END_IF

(***** DONE *****)
ST170_RFID_e.DONE: (* Letzter Schritt  *)
    IF NOT xIN_AlarmAktiv THEN
        //AUTO
        IF (enIN_State = StateAUTO) AND xIN_RestartCYCL THEN
            iOUT_Step := ST170_RFID_e.START;
            //STEP / END / LEERFAHREN restart
        ELSIF (enIN_State < StateAUTO) AND (enIN_State >= enState.StateSTEP) AND xIN_RestartCYCL THEN
            iOUT_Step := ST170_RFID_e.START;
            //STEP / END / LEERFAHREN fertig
        ELSIF (enIN_State = StateREADY) THEN
            iOUT_Step := ST170_RFID_e.READY;
        END_IF;
    END_IF;

(************ ERROR *************)
ST170_RFID_e.ERROR: (* ERROR *) ;

END_CASE;

END_FUNCTION_BLOCK

// ---- POUs/20_AUTO/ST175/FB_AUT_175.TcPOU
FUNCTION_BLOCK FB_AUT_175 EXTENDS FB_AUT_ABSTRACT
(****************************************************************************)
(*	POU_AUT_zxx			Bausteinaufrufe Station	zxx							*)
(*	Status				ungetestet											*)
(*  Version:			1.0													*)
(*	Beschrieb:																*)
(*																			*)
(*	Abläufe:			FB_ABLzxxA		Hauptablauf							*)
(*																			*)
(*																			*)
(* 	25.09.2019/Dj															*)
(****************************************************************************)
(*	dd.mm.yyyy   KZ    x.y			Beschrieb								*)
(****************************************************************************)
VAR_INPUT

    (* spezifische Eingänge *)

END_VAR
VAR_OUTPUT

    (* spezifische Ausgänge *)

END_VAR
VAR
    (* Bausteine *)
    fb_laser : FB_ABL_175;

    fb_stat : FB_AUT_Statistics;

END_VAR

(*******************************************************************)
(* Timer *)
(*******************************************************************)

(*******************************************************************)
(* Flanken / Merker *)
(*******************************************************************)
//MANU CYCLE
IF (enIN_State = StateMANU) AND xIN_ManuCycle THEN
    xManuCycle := TRUE;
END_IF;

IF (enIN_State <> StateMANU) OR xOUT_Done THEN
    xManuCycle := FALSE;
END_IF

//NEXT STEP
xNextStep := (enIN_State > StateSTEP) OR
             ((enIN_State = StateSTEP) AND xIN_Step) OR
             ((enIN_State = StateMANU) AND xManuCycle);

//RESET
xReset := (enIN_State < StateREADY) AND (enIN_State <> StateINIT) AND NOT xManuCycle;

(*******************************************************************)
(* Bausteinaufrufe Abläufe *)
(*******************************************************************)

xRelease := MAIN.MoverMan.IsProcessUsed(THIS^);

fb_laser(xIN_Reset       := xReset,
         xIN_Init        := xIN_Init,
         xIN_Quit        := xIN_Quit,
         xIN_Start       := enIN_State >= enState.StateLEER AND xRelease,
         xIN_Sperre      := NOT xIN_On,
         xIN_NextStep    := xNextStep,
         xIN_AlarmAktiv  := xIN_AlarmAktiv,
         xIN_DryCycle    := xIN_DryCycle,
         xIN_RestartCYCL := enIN_State >= enState.StateLEER,
         enIN_State      := enIN_State,
         tIN_Timeout     := tIN_Timeout,
         pxFG_Freigabe   := ADR(xRelease),
         // CleverTrackLib
         Mover := THIS^.Mover);

fb_stat(xIN_Enable  := enState.StateAUTO = enIN_State,
        xIN_Waiting := fb_laser.xOUT_Wait,
        xIN_Running := (fb_laser.iOUT_Step >= ST175_LASER_e.START) AND
                       (fb_laser.iOUT_Step <= ST175_LASER_e.DONE),
        // Since we use a mover system, a cycle is done when we are waiting on a mover
        xIN_Done := fb_laser.iOUT_Step = ST175_LASER_e.waitOnMover);

(*******************************************************************)
(* Bausteinaufruf Error Station *)
(*******************************************************************)
// POU_ERR_VORLAGE(xIN_QUIT := xIN_Quit, pstrArIN_ALARM := ADR(HMI.strArALARM[1]));

(*******************************************************************)
(* OUTPUT *)
(*******************************************************************)
xOUT_InitDone := fb_laser.xOUT_InitDone;
xOUT_Ready    := fb_laser.xOUT_Ready;
xOUT_Done     := fb_laser.xOUT_Done;
xOUT_ErrFlag  := fb_laser.xOUT_ErrFlag;
xOUT_Wait     := fb_laser.xOUT_Wait;
xOUT_AlarmST  := xOUT_ErrFlag;

(* % of completion of the process *)
PROPERTY iCompletionPC : INT
GET
iCompletionPC := THIS^.fb_laser.iOUT_ProcessCompletion;
END_GET
END_PROPERTY

PROPERTY ProcessExecution : ProcessExecution_e
GET
ProcessExecution := THIS^._ProcessExecution;
END_GET
SET
THIS^._ProcessExecution := ProcessExecution;
END_SET
END_PROPERTY

PROPERTY xBusy : BOOL
GET
xBusy := THIS^.fb_laser.xOUT_Busy;
END_GET
SET
END_SET
END_PROPERTY

PROPERTY xDone : BOOL
GET
xDone := THIS^.fb_laser.xOUT_Ready OR THIS^.fb_laser.xOUT_Done;
END_GET
END_PROPERTY

PROPERTY xMoverPathFree : BOOL
GET
xMoverPathFree := THIS^.fb_laser.xOUT_MoverFree OR THIS^.fb_laser.xOUT_Ready OR THIS^.fb_laser.xOUT_Done;
END_GET
END_PROPERTY

PROPERTY xMoverShouldLeave : BOOL
GET
xMoverShouldLeave := THIS^.fb_laser.iOUT_Step = ST175_LASER_e.SYNC_MOVER_LEAVE;
END_GET
END_PROPERTY

END_FUNCTION_BLOCK

// ---- POUs/20_AUTO/ST175/FB_ABL_175.TcPOU
FUNCTION_BLOCK FB_ABL_175
(****************************************************************************************)
(*	TITEL				laden kristall- Modul	    										*)
(*	Status				ungetestet                         								*)
(*	Beschrieb:			Ablaufbeschreibung												*)
(*																						*)
(*	Steps:	self-explained using enum													*)
(***********************************Revisionen*******************************************)
(*	see github blames																	*)
(****************************************************************************************)

VAR_INPUT
    xIN_Reset       : BOOL;          // Schrittkette zurücksetzen 
    xIN_Init        : BOOL;          // Initialisieren
    xIN_Quit        : BOOL;          // Fehler quittieren 
    xIN_Start       : BOOL;          // Startbefehl
    xIN_Sperre      : BOOL;          // FB Sperren 
    xIN_NextStep    : BOOL;          // Nächsten Schritt ausführen 
    xIN_AlarmAktiv  : BOOL;          // Anlage hat Alarm
    xIN_DryCycle    : BOOL;          // Fahren ohne Teile
    xIN_RestartCYCL : BOOL;          // Zyklus erneut starten im STEP, END, LEERFAHREN
    enIN_State      : enState;       // Status Anlage
    tIN_Timeout     : TIME := T#10s; // Timout

    pxFG_Freigabe : POINTER TO BOOL; //Freigabe von Station

    // Application specific
    Mover : REFERENCE TO FB_Mover;

END_VAR
VAR_OUTPUT
    (* standart Ausgänge *)
    xOUT_ErrFlag  : BOOL;          // Error Flag 
    xOUT_Busy     : BOOL;          // Baustein befindet sich im Ablauf 
    xOUT_Done     : BOOL;          // Baustein hat den Ablauf beendet 		
    xOUT_Ready    : BOOL;          // Ready to begin, should be the same state as done	
    xOUT_Timeout  : BOOL;          // Timeout FB 
    xOUT_InitDone : BOOL;          // initialisierung fertig
    xOUT_Wait     : BOOL;          // Wartet auf Bedingung
    iOUT_Step     : ST175_LASER_e; // Aktueller Schritt 
    sOUT_Step     : STRING;        // Aktueller Schritt but in string format
    bOUT_Error    : BYTE;          // Fehlernummer

    iOUT_ProcessCompletion : INT;  //process completion, express in % (0-100)
    xOUT_MoverFree         : BOOL; // The mover is free to move
END_VAR
VAR
    (* Standard *)
    (* Schritt *)
    iLastStep : ST175_LASER_e; // Merker letzter Schritt 
    iPreStep  : ST175_LASER_e; // Schritt zurück nach Alarm 
    iAktStep  : ST175_LASER_e; // aktueller Schritt

    // Trigger Starten 
    rtSTART : R_TRIG;
    // Timer TimeOut 
    TON_Timeout : TON;

    (* Bausteine *)
    fb_trumpf_laser : FB_Laser_ABL;

    fb_handling  : FB_ZylMo2El_V2_1;
    fb_doorEntry : FB_ZylMo2El_V2_1;
    fb_doorExit  : FB_ZylMo2El_V2_1;

    simu_handling  : FB_Simu_Zyl2Pos;
    simu_doorEntry : FB_Simu_Zyl2Pos;
    simu_doorExit  : FB_Simu_Zyl2Pos;

    (* Spezial *)
    xLASER_Result_OK  : BOOL;
    xLASER_First_mark : BOOL := FALSE;

    sErrorSuffixFileName : STRING; // suffix used to tell the user to use the file for bad pieces

END_VAR
VAR CONSTANT
    LASER_SIMULATION : BOOL := FALSE; // Set to TRUE to simulate this part of the program
END_VAR

(*******************************************************************)
(* Trigger  *)
(*******************************************************************)
(* Zurücksetzen *)
IF xIN_RESET THEN
    iPreStep  := ST175_LASER_e.RESET;
    iOUT_Step := ST175_LASER_e.RESET;
END_IF;

(* Error Quittieren *)
IF (bOUT_Error <> 0) AND xIN_Quit THEN
    xOUT_ErrFlag := FALSE;
    bOUT_Error   := 0;
    iOUT_Step    := iPreStep;
END_IF;

(*******************************************************************)
(* Timer *)
(*******************************************************************)
TON_Timeout(IN := xIN_NextStep AND (iLastStep = iOUT_Step) (*todo FG *) ,
            PT := tIN_Timeout);

(*******************************************************************)
(* Bausteine *)
(*******************************************************************)

// We manage the suffix of the laser file
IF __ISVALIDREF(Mover) AND_THEN Mover.IsPieceBad() THEN
    sErrorSuffixFileName := '_F';
ELSE
    sErrorSuffixFileName := '';
END_IF

fb_trumpf_laser(xIN_Start          := ST175_LASER_e.LASER_start = iOUT_Step,
                xIN_WarmUpLaser    := ST175_LASER_e.Init_laser_warmup = iOUT_Step,
                sIN_FileName       := CONCAT(_20_AUTO.recipe.st175.file_name, sErrorSuffixFileName),
                sIN_ErrorCode      :=, // set below
                xIN_StationInError := __ISVALIDREF(Mover) AND_THEN Mover.IsPieceBad());

// pneumatics
fb_handling(xIN_Reset    := xIN_Reset OR (ST175_LASER_e.RESET = iOUT_Step),
            xIN_Quit     := xIN_Quit,
            xIN_Manu     := enState.StateMANU = enIN_State,
            pbtIN_Button := ADR(HMI.btManuCylinders[StationList_e.ST175][1]),
            xIN_GS       := simu_handling.xOUT_inGS,
            xIN_AS       := simu_handling.xOUT_inAS,
            xIN_FREE     := TRUE,
            xINtoGS      := (ST175_LASER_e.Init_pneumatics = iOUT_Step) OR
                            (ST175_LASER_e.handling_up = iOUT_Step),
            xINtoAS   := ST175_LASER_e.handling_down = iOUT_Step,
            tIN_ErrAS := DINT_TO_TIME(_20_AUTO.recipe.cylinder2Pos[StationList_e.ST175]
                                          [ST175_Cylinders_e.Niederhalter].toAS_alarm_time),
            tIN_ErrGS := DINT_TO_TIME(_20_AUTO.recipe.cylinder2Pos[StationList_e.ST175]
                                          [ST175_Cylinders_e.Niederhalter].toGS_alarm_time),
            tIN_WaitAS := DINT_TO_TIME(_20_AUTO.recipe.cylinder2Pos[StationList_e.ST175]
                                           [ST175_Cylinders_e.Niederhalter].toAS_wait_time),
            tIN_WaitGS := DINT_TO_TIME(_20_AUTO.recipe.cylinder2Pos[StationList_e.ST175]
                                           [ST175_Cylinders_e.Niederhalter].toGS_wait_time));

simu_handling(xIN_Enable := TRUE, //LASER_SIMULATION AND CONST.USE_SIMULATION,
              xIN_inGS   := IO_BOX.I9300_ST175_wegmesssensor < 10,
              xIN_inAS   := IO_BOX.I9300_ST175_wegmesssensor > 200,
              xIN_valve  := fb_handling.xOUT_VALVE,
              tIN_GS_ms  := 200,  // ms
              tIN_AS_ms  := 200); // ms

fb_doorEntry(xIN_Reset    := xIN_Reset OR (ST175_LASER_e.RESET = iOUT_Step),
             xIN_Quit     := xIN_Quit,
             xIN_Manu     := enState.StateMANU = enIN_State,
             pbtIN_Button := ADR(HMI.btManuCylinders[StationList_e.ST175][2]),
             xIN_GS       := simu_doorEntry.xOUT_inGS,
             xIN_AS       := simu_doorEntry.xOUT_inAS,
             xIN_FREE     := TRUE,
             xINtoGS      := (ST175_LASER_e.Init_pneumatics = iOUT_Step) OR
                             (ST175_LASER_e.open_doors = iOUT_Step),
             xINtoAS   := ST175_LASER_e.close_doors = iOUT_Step,
             tIN_ErrAS := DINT_TO_TIME(_20_AUTO.recipe.cylinder2Pos[StationList_e.ST175]
                                           [ST175_Cylinders_e.Door_entry].toAS_alarm_time),
             tIN_ErrGS := DINT_TO_TIME(_20_AUTO.recipe.cylinder2Pos[StationList_e.ST175]
                                           [ST175_Cylinders_e.Door_entry].toGS_alarm_time),
             tIN_WaitAS := DINT_TO_TIME(_20_AUTO.recipe.cylinder2Pos[StationList_e.ST175]
                                            [ST175_Cylinders_e.Door_entry].toAS_wait_time),
             tIN_WaitGS := DINT_TO_TIME(_20_AUTO.recipe.cylinder2Pos[StationList_e.ST175]
                                            [ST175_Cylinders_e.Door_entry].toGS_wait_time));

simu_doorEntry(xIN_Enable := TRUE,  //LASER_SIMULATION AND CONST.USE_SIMULATION,
               xIN_inGS   := FALSE, // no sensor here
               xIN_inAS   := FALSE, // no sensor here
               xIN_valve  := fb_doorEntry.xOUT_VALVE,
               tIN_GS_ms  := 400,  // ms
               tIN_AS_ms  := 400); // ms

fb_doorExit(xIN_Reset    := xIN_Reset OR (ST175_LASER_e.RESET = iOUT_Step),
            xIN_Quit     := xIN_Quit,
            xIN_Manu     := enState.StateMANU = enIN_State,
            pbtIN_Button := ADR(HMI.btManuCylinders[StationList_e.ST175][3]),
            xIN_GS       := simu_doorExit.xOUT_inGS,
            xIN_AS       := simu_doorExit.xOUT_inAS,
            xIN_FREE     := TRUE,
            xINtoGS      := (ST175_LASER_e.Init_pneumatics = iOUT_Step) OR
                            (ST175_LASER_e.open_doors = iOUT_Step),
            xINtoAS   := ST175_LASER_e.close_doors = iOUT_Step,
            tIN_ErrAS := DINT_TO_TIME(_20_AUTO.recipe.cylinder2Pos[StationList_e.ST175]
                                          [ST175_Cylinders_e.Door_exit].toAS_alarm_time),
            tIN_ErrGS := DINT_TO_TIME(_20_AUTO.recipe.cylinder2Pos[StationList_e.ST175]
                                          [ST175_Cylinders_e.Door_exit].toGS_alarm_time),
            tIN_WaitAS := DINT_TO_TIME(_20_AUTO.recipe.cylinder2Pos[StationList_e.ST175]
                                           [ST175_Cylinders_e.Door_exit].toAS_wait_time),
            tIN_WaitGS := DINT_TO_TIME(_20_AUTO.recipe.cylinder2Pos[StationList_e.ST175]
                                           [ST175_Cylinders_e.Door_exit].toGS_wait_time));

simu_doorExit(xIN_Enable := TRUE,  //LASER_SIMULATION AND CONST.USE_SIMULATION,
              xIN_inGS   := FALSE, // no sensor here
              xIN_inAS   := FALSE, // no sensor here
              xIN_valve  := fb_doorExit.xOUT_VALVE,
              tIN_GS_ms  := 400,  // ms
              tIN_AS_ms  := 400); // ms

(*******************************************************************)
(* OUTPUTS *)
(*******************************************************************)
// Error Flag 
xOUT_ErrFlag := (bOUT_Error <> 0) OR (ST175_LASER_e.ERROR = iOUT_Step);
// Baustein befindet sich im Ablauf 
xOUT_Busy := (iOUT_Step > ST175_LASER_e.READY) AND (iOUT_Step < ST175_LASER_e.DONE);
// Baustein hat den Ablauf beendet
xOUT_Done := (iOUT_Step = ST175_LASER_e.DONE);
// Process ready
xOUT_Ready := (iOUT_Step = ST175_LASER_e.READY) OR (iOUT_Step = ST175_LASER_e.waitOnMover);
// Timeout FB 				 		
xOUT_Timeout := TON_Timeout.Q;
// Itialisierung fertig			
xOUT_InitDone := (iOUT_Step = ST175_LASER_e.READY) OR (iOUT_Step = ST175_LASER_e.waitOnMover);
// Aktueller Schritt			
iOUT_Step := iOUT_Step; //Im Ablauf gesetzt		
sOUT_Step := TO_STRING(iOUT_Step);
//Fehlernummer	 
bOUT_Error := bOUT_Error; //Im Ablauf/FB gesetzt	
(* Warte (alle Schritte wo auf FG oder Teile gewartet wird) *)
xOUT_Wait := (iOUT_Step = ST175_LASER_e.DONE) OR
             (iOUT_Step = ST175_LASER_e.READY) OR
             (iOUT_Step = ST175_LASER_e.START) OR
             (iOUT_Step = ST175_LASER_e.waitOnMover) OR
             (iOUT_Step = ST175_LASER_e.SYNC_MOVER_LEAVE);

xOUT_MoverFree := fb_handling.xOUT_inGS AND fb_doorEntry.xOUT_inGS AND fb_doorExit.xOUT_inGS;

iOUT_ProcessCompletion := F_GetPercent_2(iAktStep,
                                         iAktStep,
                                         iAktStep,
                                         ST175_LASER_e.close_doors,
                                         ST175_LASER_e.SYNC_MOVER_LEAVE);

(* BIG CHANGE IN OUTPUT, PLEASE UPDATE *)
IO_BOX.Q5300_14_ST175_niederhalter :=
    fb_doorEntry.xOUT_VALVE AND NOT (LASER_SIMULATION AND CONST.USE_SIMULATION);

IO_BOX.Q5301_14_ST175_kabinentur_einlaufseite :=
    fb_doorExit.xOUT_VALVE AND NOT (LASER_SIMULATION AND CONST.USE_SIMULATION);

IO_BOX.Q5302_14_ST175_kabinentur_auflaufseite :=
    fb_handling.xOUT_VALVE AND NOT (LASER_SIMULATION AND CONST.USE_SIMULATION);

OUT.Q101_ST175_Sauger_LN_230_Start :=
    (enIN_State >= enState.StateEND) AND
    (iOUT_Step > ST175_LASER_e.close_doors) AND
    (iOUT_Step <= ST175_LASER_e.open_doors) AND
    NOT (LASER_SIMULATION AND CONST.USE_SIMULATION);

(*******************************************************************)
(* Ablauf *)
(*******************************************************************)

(* Sperren *)
IF xIN_Sperre THEN
    iPreStep  := ST175_LASER_e.RESET;
    iOUT_Step := ST175_LASER_e.RESET;
    RETURN;
END_IF;

(* Schritt Merker *)
IF iAktStep <> iOUT_Step THEN
    iLastStep := iAktStep;
    iAktStep  := iOUT_Step;
END_IF

(* START *)
rtSTART(CLK := xIN_Start);

IF 0 = bOUT_Error THEN
    IF fb_handling.xOUT_ErrFlag THEN
        bOUT_Error := 11;
    ELSIF fb_doorEntry.xOUT_ErrFlag THEN
        bOUT_Error := 12;
    ELSIF fb_doorExit.xOUT_ErrFlag THEN
        bOUT_Error := 13;
    ELSIF fb_trumpf_laser.xOUT_ERROR THEN
        bOUT_Error := 20;
    END_IF
ELSIF iOUT_Step < ST175_LASER_e.ERROR THEN
    iOUT_Step := ST175_LASER_e.ERROR;
END_IF

(*******************************************************************)
(* Schrittkette  *)
(*******************************************************************)
CASE iOUT_Step OF

(***** RESET *****)
ST175_LASER_e.RESET: (* Schritt 0-99 *)
    //Initialisierungen
    //Start Init Ablauf
    IF xIN_Init THEN
        iOUT_Step := ST175_LASER_e.INIT;
        //Start Manu Ablauf
    ELSIF enIN_State = StateMANU AND xIN_NextStep THEN
        iOUT_Step := ST175_LASER_e.INIT;
    END_IF;

(***** INIT *****)
ST175_LASER_e.INIT: (* Grundstellung ? *)
    iOUT_Step := ST175_LASER_e.Init_pneumatics;

ST175_LASER_e.Init_pneumatics:
    IF fb_handling.xOUT_inGS AND fb_doorEntry.xOUT_inGS AND fb_doorExit.xOUT_inGS THEN
        iOUT_Step := ST175_LASER_e.Init_laser_warmup;
    END_IF

ST175_LASER_e.Init_laser_warmup:
    iOUT_Step := ST175_LASER_e.READY;

(***** READY / INIT DONE *****)
ST175_LASER_e.READY:  (* Start AUTO,END,LEER,STEP *)
    IF xIN_Start THEN //IF rtSTART.Q THEN
        iOUT_Step := ST175_LASER_e.START;
    END_IF

(***** START  ZYKLISCH *****)
ST175_LASER_e.START: (*  *)
    IF xIN_NextStep AND pxFG_Freigabe^ THEN
        iOUT_Step        := ST175_LASER_e.waitOnMover;
        iPreStep         := ST175_LASER_e.waitOnMover;
        xLASER_Result_OK := FALSE;
    END_IF;

ST175_LASER_e.waitOnMover: (*  *)
    IF xIN_NextStep AND __ISVALIDREF(Mover) THEN
        IF (Mover.GetLastStationDone() >= 175) THEN
            iOUT_Step := ST175_LASER_e.SYNC_MOVER_LEAVE;
        ELSIF Mover.GetLastStationDone() < INT#150 THEN
            iOUT_Step := ST175_LASER_e.SYNC_MOVER_LEAVE;
        ELSE
            IF NOT MAIN.MoverMan.IsMoverInRange(from_pos := 7750.0, to_pos := 8050.0) THEN
                iOUT_Step := ST175_LASER_e.close_doors;
            END_IF
        END_IF
    END_IF;

ST175_LASER_e.close_doors:
    IF fb_doorEntry.xOUT_inAS AND fb_doorExit.xOUT_inAS THEN
        xLASER_First_mark := FALSE;
        iOUT_Step         := ST175_LASER_e.handling_down;
    END_IF

ST175_LASER_e.handling_down:
    IF fb_handling.xOUT_inAS THEN
        IF LASER_SIMULATION AND CONST.USE_SIMULATION THEN
            iOUT_Step := ST175_LASER_e.handling_up;
        ELSE
            iOUT_Step := ST175_LASER_e.LASER_start;
        END_IF
    END_IF

ST175_LASER_e.LASER_start:
    IF fb_trumpf_laser.xOUT_BUSY THEN
        IF __ISVALIDREF(Mover) THEN

            IF NOT _20_AUTO.recipe.st175.isTypeSmartOrMini THEN
                fb_trumpf_laser.sIN_ErrorCode := Mover.GetErrorCode();
            ELSIF NOT xLASER_First_mark THEN
                fb_trumpf_laser.sIN_ErrorCode := CONCAT('R-', Mover.GetErrorCode());
            ELSE
                fb_trumpf_laser.sIN_ErrorCode := CONCAT('L-', Mover.GetErrorCode());
            END_IF

            IF NOT Mover.SetLastStation(175) THEN
                ASSERT(0);
            END_IF
        END_IF

        iOUT_Step := ST175_LASER_e.LASER_wait_on_finish;
    END_IF

ST175_LASER_e.LASER_wait_on_finish:
    IF fb_trumpf_laser.xOUT_DONE OR NOT fb_trumpf_laser.xOUT_BUSY THEN
        iOUT_Step        := ST175_LASER_e.handling_up;
        xLASER_Result_OK := NOT fb_trumpf_laser.xOUT_ERROR;
    END_IF

ST175_LASER_e.handling_up:
    IF fb_handling.xOUT_inGS THEN
        IF NOT _20_AUTO.recipe.st175.isTypeSmartOrMini OR xLASER_First_mark THEN
            iOUT_Step := ST175_LASER_e.open_doors;
        ELSE
            iOUT_Step := ST175_LASER_e.move_shuttle_to_left_piece;
        END_IF
    END_IF

ST175_LASER_e.move_shuttle_to_left_piece:
    IF xIN_NextStep AND __ISVALIDREF(Mover) AND_THEN Mover.MoveRelativeInsideStation(118.0) THEN
        iOUT_Step := ST175_LASER_e.wait_shuttle_in_place;
        iPreStep  := ST175_LASER_e.handling_down;
    END_IF

ST175_LASER_e.wait_shuttle_in_place:
    IF xIN_NextStep AND __ISVALIDREF(Mover) AND_THEN Mover.IsInStationPos() THEN
        xLASER_First_mark := TRUE;
        iOUT_Step         := ST175_LASER_e.handling_down;
    END_IF

ST175_LASER_e.open_doors:
    IF fb_doorEntry.xOUT_inGS AND fb_doorExit.xOUT_inGS THEN
        iOUT_Step := ST175_LASER_e.SYNC_MOVER_LEAVE;

        IF __ISVALIDREF(Mover) AND NOT xLASER_Result_OK THEN
            Mover.SetErrorCode('175-B');

            IF NOT Mover.SetLastStation(-175) THEN
                ASSERT(0);
            END_IF
        ELSIF __ISVALIDREF(Mover) AND xLASER_Result_OK THEN
            IF NOT Mover.SetLastStation(175) THEN
                ASSERT(0);
            END_IF
        END_IF
    END_IF

ST175_LASER_e.SYNC_MOVER_LEAVE:
    // The mover needs to be taken by MoverMan
    IF NOT __ISVALIDREF(Mover) THEN
        iOUT_Step := ST175_LASER_e.DONE;
    END_IF

(***** DONE *****)
ST175_LASER_e.DONE: (* Letzter Schritt  *)
    IF NOT xIN_AlarmAktiv THEN
        //AUTO
        IF (enIN_State = StateAUTO) AND xIN_RestartCYCL THEN
            iOUT_Step := ST175_LASER_e.START;
            //STEP / END / LEERFAHREN restart
        ELSIF (enIN_State < StateAUTO) AND (enIN_State >= enState.StateSTEP) AND xIN_RestartCYCL THEN
            iOUT_Step := ST175_LASER_e.START;
            //STEP / END / LEERFAHREN fertig
        ELSIF (enIN_State = StateREADY) THEN
            iOUT_Step := ST175_LASER_e.READY;
        END_IF;
    END_IF;

(************ ERROR *************)
ST175_LASER_e.ERROR: (* ERROR *) ;

END_CASE;

END_FUNCTION_BLOCK

// ---- POUs/20_AUTO/ST175/Trumpf/FB_Laser_ABL.TcPOU
FUNCTION_BLOCK FB_Laser_ABL
VAR_INPUT
    xIN_Start          : BOOL;
    xIN_WarmUpLaser    : BOOL; // activate laser, only possible when cycle is not started
    sIN_FileName       : STRING := 'Someting here please';
    xIN_ResetData      : BOOL;       // reset all data, used to ensure that the marking data are in the laser
    sIN_ErrorCode      : STRING(NUM_STRING_LENGTH); // error code to write when a station is in error
    xIN_StationInError : BOOL;       // don't write normal data, write error data instead
END_VAR
VAR_OUTPUT
    xOUT_DONE  : BOOL;
    xOUT_ERROR : BOOL;
    xOUT_BUSY  : BOOL;
END_VAR
VAR
    iStep     : INT := 0;
    sDataTime : STRING(NUM_STRING_LENGTH);

    sLastName : STRING;     // var used to see if last value has changed or not
    sLastNum  : STRING(NUM_STRING_LENGTH); // var used to see if last value has changed or not

    fb_time : NT_GetTime;
END_VAR
VAR CONSTANT
	NUM_STRING_LENGTH : UDINT := 32; // maximum string length for the number
END_VAR

fb_time(NETID := '',
        START :=,
        TMOUT := T#1S);

IF xIN_ResetData THEN
    MEMSET(ADR(sLastName), 0, SIZEOF(sLastName));
    MEMSET(ADR(sLastNum), 0, SIZEOF(sLastNum));
END_IF

IF 0 = iStep AND xIN_WarmUpLaser AND if_SingleCmds.bReady THEN
    if_SingleCmds.iStepNr := 10; // TLV - Activate Laser / Open Shutter
    if_SingleCmds.bStart  := TRUE;
END_IF

CASE iStep OF

0: (* wait on start *)
    IF xIN_Start THEN
        iStep := 1000;
    END_IF

1000: (* TruMark *)
    IF if_SingleCmds.bReady THEN
        IF if_TruMark.Status.b6_LaserMalfunction THEN
            if_SingleCmds.iStepNr := 120; // TLV - Activate Laser / Open Shutter
            if_SingleCmds.bStart  := TRUE;
            iStep                 := 1010;
        ELSIF if_TruMark.Status.b0_Laser_On THEN
            iStep := 1040; // go to get the time
        ELSE
            iStep := 1020;
        END_IF;
    END_IF

1010: (* Reset Done*)
    IF if_SingleCmds.bReady THEN
        iStep := 1020;
    END_IF

1020: (* Laser ON *)
    IF if_SingleCmds.bReady THEN
        if_SingleCmds.iStepNr := 10; // TLV - Activate Laser / Open Shutter
        if_SingleCmds.bStart  := TRUE;
        iStep                 := 1030;
    END_IF;

1030: (* ON DONE*)
    IF if_SingleCmds.bReady THEN
        iStep := 1040;
    END_IF;

1040: (* get time *)
    fb_time.START := TRUE;
    iStep         := 1050;

1050: (* get time *)
    IF NOT fb_time.BUSY THEN
        fb_time.START := FALSE;
        iStep         := 1100;
    END_IF

1100: (* New FILE ? todo *)
    IF 0 = FIND(sLastName, sIN_FileName) OR (LEN(sLastName) <> LEN(sIN_FileName)) THEN
        iStep := 1110;
    ELSIF xIN_StationInError THEN
        iStep := 1110;
    ELSE
        iStep := 1130;
    END_IF

1110: (* Load File *)
    IF if_SingleCmds.bReady THEN
        if_SingleCmds.iStepNr     := 20; // TLV - Load Marking-File with 2 variables
        if_SingleCmds.sInputValue := CONCAT('C:\Aquis\', CONCAT(sIN_FileName, '.VLF'));
        sLastName                 := sIN_FileName;

        if_SingleCmds.bStart := TRUE;
        iStep                := 1120;
    END_IF

1120: (* Conversation *)
    IF if_SingleCmds.bReady THEN
        if_SingleCmds.iStepNr := 30; // TLV - Request state of conversion
        if_SingleCmds.bStart  := TRUE;
        iStep                 := 1130;
    END_IF

1130: (* New Var ? todo*)
    // date format : Y1M1D1D2M2Y2-Sx

    IF NOT xIN_StationInError THEN
        sDataTime[0] := F_ToASC(str := '0') + TO_BYTE((fb_time.TIMESTR.wYear MOD 100) / 10);  // Y1
        sDataTime[1] := F_ToASC(str := '0') + TO_BYTE((fb_time.TIMESTR.wMonth MOD 100) / 10); // M1
        sDataTime[2] := F_ToASC(str := '0') + TO_BYTE((fb_time.TIMESTR.wDay MOD 100) / 10);   // D1
        sDataTime[3] := F_ToASC(str := '0') + TO_BYTE(fb_time.TIMESTR.wDay MOD 10);           // D2
        sDataTime[4] := F_ToASC(str := '0') + TO_BYTE(fb_time.TIMESTR.wMonth MOD 10);         // M2
        sDataTime[5] := F_ToASC(str := '0') + TO_BYTE(fb_time.TIMESTR.wYear MOD 10);          // Y2
        sDataTime[6] := F_ToASC(str := '-');
        sDataTime[7] := F_ToASC(str := 'S');
        sDataTime[8] := F_ToASC(str := '1'); // TODO, team of the day
        sDataTime[9] := 0;
    ELSE
		sDataTime := sIN_ErrorCode;
    END_IF

    IF 0 = FIND(sLastNum, sDataTime) OR
       (LEN(sLastNum) <> LEN(sDataTime)) OR
       ((sDataTime[2] = F_ToASC(str := '0')) AND (sDataTime[3] = F_ToASC(str := '0'))) THEN
        iStep := 1140;
    ELSE
        iStep := 1170;
    END_IF

    MEMCPY(ADR(sLastNum), ADR(sDataTime), NUM_STRING_LENGTH);

1140: (* Set Var *)
    IF if_SingleCmds.bReady THEN
        if_SingleCmds.iStepNr := 35; // TLV - Set Variable
        // Variable name = 'Var1'	value = '3374'		Delimiter = ; --> will be replased with 0x00 in TruMark_Ethercat
        if_SingleCmds.sInputValue := CONCAT('Var1;', TO_STRING(sDataTime));

        if_SingleCmds.bStart := TRUE;
        iStep                := 1150;
    END_IF

1150: (* Var Done -> Convert *)
    IF if_SingleCmds.bReady THEN
        if_SingleCmds.iStepNr := 55; // TLV - Convert Marking File
        if_SingleCmds.bStart  := TRUE;
        iStep                 := 1160;
    END_IF

1160: (* Request Convert *)
    IF if_SingleCmds.bReady THEN
        if_SingleCmds.iStepNr := 30; // TLV - Request state of conversion
        if_SingleCmds.bStart  := TRUE;
        iStep                 := 1170;
    END_IF

1170: (* Request State *)
    IF if_SingleCmds.bReady THEN
        if_SingleCmds.iStepNr := 40; // TLV - Request Laser state
        if_SingleCmds.bStart  := TRUE;
        iStep                 := 1200;
    END_IF

1200: (* mark *)
    IF if_TruMark.Status.b0_Laser_On AND if_TruMark.Status.b1_Laser_Ready AND if_SingleCmds.bReady THEN
        if_SingleCmds.iStepNr := 50; // TLV - Activate Laser / Open Shutter
        if_SingleCmds.bStart  := TRUE;
        iStep                 := 1210;
    END_IF

// is done when safety signals are FALSE
// 1210: (* release laser *)
//     IF if_SingleCmds.bReady THEN
//         if_SingleCmds.iStepNr := 12; // TLV - Desactivate Laser
//         if_SingleCmds.bStart  := TRUE;
//         iStep                 := 1300;
//     END_IF

1210:
    IF if_TruMark.Status.b15_Mark_Active THEN
        iStep := 1220;
    END_IF

1220:
    IF NOT if_TruMark.Status.b15_Mark_Active THEN
        iStep := 1300;
    END_IF

1300: (* Check GS Datumsringüberwachung *)
    IF NOT xIN_Start THEN
        iStep := 0;
    END_IF

END_CASE

xOUT_DONE  := 1300 = iStep;
xOUT_BUSY  := (iStep >= 1000 AND iStep < 1300) OR NOT if_SingleCmds.bReady;
xOUT_ERROR := if_TruMark.bError;

END_FUNCTION_BLOCK

// ---- POUs/20_AUTO/ST100/FB_AUT_MODIFY.TcPOU
FUNCTION_BLOCK FB_AUT_MODIFY EXTENDS FB_AUT_ABSTRACT IMPLEMENTS ISimuMoverTimers
    (****************************************************************************)
    (*	POU_AUT_zxx			Bausteinaufrufe Station	zxx							*)
    (*	Status				ungetestet											*)
    (*  Version:			1.0													*)
    (*	Beschrieb:																*)
    (*																			*)
    (*	Abläufe:			FB_ABLzxxA		Hauptablauf							*)
    (*																			*)
    (*																			*)
    (* 	25.09.2019/Dj															*)
    (****************************************************************************)
    (*	dd.mm.yyyy   KZ    x.y			Beschrieb								*)
    (****************************************************************************)
VAR_INPUT
    (* spezifische Eingänge *)

END_VAR
VAR_OUTPUT
    (* spezifische Ausgänge *)

END_VAR
VAR
    (* Bausteine *)
    _FB_ABL_100A : FB_ABL_MODIFY;
END_VAR

(*******************************************************************)
(* Timer *)
(*******************************************************************)

(*******************************************************************)
(* Flanken / Merker *)
(*******************************************************************)
//MANU CYCLE
IF (enIN_State = StateMANU) AND xIN_ManuCycle THEN
    xManuCycle := TRUE;
END_IF;

IF (enIN_State <> StateMANU) OR xOUT_Done THEN
    xManuCycle := FALSE;
END_IF

//NEXT STEP
xNextStep := (enIN_State > StateSTEP) OR
             ((enIN_State = StateSTEP) AND xIN_Step) OR
             ((enIN_State = StateMANU) AND xManuCycle);

//RESET
xReset := (enIN_State < StateREADY) AND (enIN_State <> StateINIT) AND NOT xManuCycle;

(*******************************************************************)
(* Bausteinaufrufe Abläufe *)
(*******************************************************************)

_FB_ABL_100A(xIN_Reset    := xReset,
             xIN_Init     := xIN_Init,
             xIN_Quit     := xIN_Quit,
             xIN_Start    := enIN_State = enState.StateAUTO, //AND _FB_ABL_100A.xOUT_Done AND _FB_ABL_100A.xOUT_Ready,
             xIN_Sperre   := NOT xIN_On,
             xIN_NextStep := xNextStep,
             xIN_AlarmAktiv
                 := xIN_AlarmAktiv,
             xIN_DryCycle    := xIN_DryCycle,
             xIN_RestartCYCL := enIN_State = enState.StateAUTO, // only restart when the mover has move out
             enIN_State      := enIN_State,
             tIN_Timeout     := tIN_Timeout,
             pxFG_Freigabe   := ADR(xRelease),
             Mover           := THIS^.Mover,
             xOUT_ErrFlag    =>,
             xOUT_Busy       =>,
             xOUT_Done       =>,
             xOUT_Timeout    =>,
             xOUT_InitDone   =>,
             xOUT_Wait       =>,
             iOUT_Step       =>,
             bOUT_Error      =>);

(*******************************************************************)
(* Mover reset flags *)
(*******************************************************************)

(*******************************************************************)
(* OUTPUT *)
(*******************************************************************)
xOUT_InitDone := _FB_ABL_100A.xOUT_InitDone;
xOUT_Ready    := xOUT_InitDone;
xOUT_Done     := _FB_ABL_100A.xOUT_Done;
xOUT_ErrFlag  := _FB_ABL_100A.xOUT_ErrFlag;
xOUT_Wait     := _FB_ABL_100A.xOUT_Wait;
xOUT_AlarmST  := xOUT_ErrFlag;

(*******************************************************************)
(* Bausteinaufruf Error Station *)
(*******************************************************************)
// POU_ERR_VORLAGE(xIN_QUIT:=xIN_Quit , pstrArIN_ALARM:=ADR(HMI.strArALARM[1]));

METHOD GiveMover : IProcessSampleMover
VAR_INPUT
	mover : REFERENCE TO FB_Mover;
END_VAR
IF __ISVALIDREF(mover) THEN
    THIS^.Mover                       REF= mover;
END_IF
END_METHOD

(* % of completion of the process *)
PROPERTY iCompletionPC : INT
GET
iCompletionPC := THIS^._FB_ABL_100A.iOUT_ProcessCompletion;
END_GET
END_PROPERTY

(* Process time, expressed in milisecond *)
PROPERTY iProcessTimeMili_1 : DINT
GET
iProcessTimeMili_1 := TO_DINT(this^._FB_ABL_100A.iProcessTimeMili1);
END_GET
SET
THIS^._FB_ABL_100A.iProcessTimeMili1 := TO_UDINT(iProcessTimeMili_1);
END_SET
END_PROPERTY

(* Process time, expressed in milisecond *)
PROPERTY iProcessTimeMili_2 : DINT
GET
iProcessTimeMili_2 := TO_DINT(this^._FB_ABL_100A.iProcessTimeMili2);
END_GET
SET
THIS^._FB_ABL_100A.iProcessTimeMili2 := TO_UDINT(iProcessTimeMili_2);
END_SET
END_PROPERTY

PROPERTY ProcessExecution : ProcessExecution_e
GET
ProcessExecution := THIS^._ProcessExecution;
END_GET
SET
THIS^._ProcessExecution := ProcessExecution;
END_SET
END_PROPERTY

METHOD TakeMover : IProcessSampleMover
VAR_INPUT
END_VAR
THIS^.Mover REF= 0;
END_METHOD

PROPERTY xBusy : BOOL
GET
xBusy := This^._FB_ABL_100A.xOUT_Busy;
END_GET
SET
END_SET
END_PROPERTY

PROPERTY xDone : BOOL
GET
xDone := THIS^._FB_ABL_100A.xOUT_Ready OR THIS^._FB_ABL_100A.xOUT_Done;
END_GET
END_PROPERTY

PROPERTY xMoverPathFree : BOOL
GET
xMoverPathFree := THIS^._FB_ABL_100A.xOUT_MoverFree OR THIS^._FB_ABL_100A.xOUT_Ready OR THIS^._FB_ABL_100A.xOUT_Done;
END_GET
END_PROPERTY

PROPERTY xMoverShouldLeave : BOOL
GET
xMoverShouldLeave := THIS^._FB_ABL_100A.iOUT_Step = ST100_Modify_e.SYNC_MOVER_LEAVE;
END_GET
END_PROPERTY

END_FUNCTION_BLOCK

// ---- POUs/20_AUTO/ST100/FB_ABL_MODIFY.TcPOU
FUNCTION_BLOCK FB_ABL_MODIFY
(****************************************************************************************)
(*	TITEL				Bezeichnung Ablauf	    										*)
(*	Status				ungetestet                         								*)
(*  Version:			1.0																*)
(*	Beschrieb:			Ablaufbeschreibung												*)
(*																						*)
(*	Steps:																				*)
(*		RESET:=0		Reset der Station												*)
(* 		INIT:=100		Initialisieren													*)
(*		... 			...																*)
(*		READY:=999		Initialisiert, Bereit für Start									*)
(*		START:=1000		Start Zyklisch 													*)
(*		... 			...																*)
(*		DONE:=8000		Letzer Schritt													*)
(*		ERROR:=9000		ALARM/Fehler													*)
(* 	09.09.2019/Dj																		*)
(***********************************Revisionen*******************************************)
(*	dd.mm.yyyy   KZ    x.y			Beschrieb											*)
(****************************************************************************************)

VAR_INPUT
    xIN_Reset       : BOOL;          // Schrittkette zurücksetzen 
    xIN_Init        : BOOL;          // Initialisieren
    xIN_Quit        : BOOL;          // Fehler quittieren 
    xIN_Start       : BOOL;          // Startbefehl
    xIN_Sperre      : BOOL;          // FB Sperren 
    xIN_NextStep    : BOOL;          // Nächsten Schritt ausführen 
    xIN_AlarmAktiv  : BOOL;          // Anlage hat Alarm
    xIN_DryCycle    : BOOL;          // Fahren ohne Teile
    xIN_RestartCYCL : BOOL;          // Zyklus erneut starten im STEP, END, LEERFAHREN
    enIN_State      : enState;       // Status Anlage
    tIN_Timeout     : TIME := T#10s; // Timout

    pxFG_Freigabe : POINTER TO BOOL; //Freigabe von Station

    // Application specific
    iProcessTimeMili1 : UDINT := 5000; // user defined station duration, in milisecond
    iProcessTimeMili2 : UDINT := 5000; // user defined station duration, in milisecond
    Mover            : REFERENCE TO FB_Mover;
    //xIN_MoverInPos  : BOOL;          // Set this flag when a mover is in position and ready to be handled
END_VAR
VAR_OUTPUT
    (* standart Ausgänge *)
    xOUT_ErrFlag     : BOOL;   // Error Flag 
    xOUT_Busy        : BOOL;   // Baustein befindet sich im Ablauf 
    xOUT_Done        : BOOL;   // Baustein hat den Ablauf beendet 		
    xOUT_Ready       : BOOL;   // Ready to begin, should be the same state as done	
    xOUT_Timeout     : BOOL;   // Timeout FB 
    xOUT_InitDone    : BOOL;   // initialisierung fertig
    xOUT_Wait        : BOOL;   // Wartet auf Bedingung
    iOUT_Step        : INT;    // Aktueller Schritt 
    sOUT_Step        : STRING; // Aktueller Schritt but in string format
    bOUT_Error       : BYTE;   // Fehlernummer

    xOUT_MoverFree   : BOOL;   // The mover is free to move
    //xOUT_MoverNeeded : BOOL;   // A mover is needed by this station to continue its process
    iOUT_ProcessCompletion : INT; //process completion, express in % (0-100)
END_VAR
VAR
    (* Standard *)
    (* Schritt *)
    iLastStep : INT; // Merker letzter Schritt 
    iPreStep  : INT; // Schritt zurück nach Alarm 
    iAktStep  : INT; // aktueller Schritt

    // Trigger Starten 
    rtSTART : R_TRIG;
    // Timer TimeOut 
    TON_Timeout : TON;

    (* Bausteine *)

    (* Spezial *)
    iStartProcessTimeMili : UDINT; // start of the processing time, accurate at 100ns 
	
	_bBewegung : BOOL;
	_bBewegungDist : INT := 20;

END_VAR
VAR CONSTANT
END_VAR

(*******************************************************************)
(* Trigger  *)
(*******************************************************************)
(* Zurücksetzen *)
IF xIN_RESET THEN
    iPreStep  := ST100_Modify_e.RESET;
    iOUT_Step := ST100_Modify_e.RESET;
END_IF;

(* Error Quittieren *)
IF (bOUT_Error <> 0) AND xIN_Quit THEN
    xOUT_ErrFlag := FALSE;
    bOUT_Error   := 0;
    iOUT_Step    := iPreStep;
END_IF;

(*******************************************************************)
(* Timer *)
(*******************************************************************)
TON_Timeout(IN := xIN_NextStep AND (iLastStep = iOUT_Step) (*todo FG *) ,
            PT := tIN_Timeout);

(*******************************************************************)
(* Bausteine *)
(*******************************************************************)

(*******************************************************************)
(* OUTPUTS *)
(*******************************************************************)
// Error Flag 
xOUT_ErrFlag := (bOUT_Error <> 0);
// Baustein befindet sich im Ablauf 
xOUT_Busy := (iOUT_Step > ST100_Modify_e.READY) AND (iOUT_Step < ST100_Modify_e.DONE);
// Baustein hat den Ablauf beendet
xOUT_Done := (iOUT_Step = ST100_Modify_e.DONE);
// Process ready
xOUT_Ready := (iOUT_Step = ST100_Modify_e.READY);
// Timeout FB 				 		
xOUT_Timeout := TON_Timeout.Q;
// Itialisierung fertig			
xOUT_InitDone := (iOUT_Step = ST100_Modify_e.READY);
// Aktueller Schritt			
iOUT_Step := iOUT_Step; //Im Ablauf gesetzt		
sOUT_Step := TO_STRING(iOUT_Step);
//Fehlernummer	 
bOUT_Error := bOUT_Error; //Im Ablauf/FB gesetzt	
(* Warte (alle Schritte wo auf FG oder Teile gewartet wird) *)
xOUT_Wait := (iOUT_Step = ST100_Modify_e.DONE);

xOUT_MoverFree := iOUT_Step = ST100_Modify_e.waitOnMover;

iOUT_ProcessCompletion := F_GetPercent(iAktStep,
                                       ST100_Modify_e.START,
                                       ST100_Modify_e.DONE,
                                       ST100_Modify_e.proceedOperation_1,
                                       ST100_Modify_e.proceedOperation_2,
                                       iStartProcessTimeMili,
                                       TO_DINT(iProcessTimeMili1),
                                       TO_DINT(iProcessTimeMili2));

(*******************************************************************)
(* Ablauf *)
(*******************************************************************)

(* Sperren *)
IF xIN_Sperre THEN
    iPreStep  := ST100_Modify_e.RESET;
    iOUT_Step := ST100_Modify_e.RESET;
    RETURN;
END_IF;

(* Schritt Merker *)
IF iAktStep <> iOUT_Step THEN
    iLastStep := iAktStep;
    iAktStep  := iOUT_Step;
END_IF

(* START *)
rtSTART(CLK := xIN_Start);

(*******************************************************************)
(* Schrittkette  *)
(*******************************************************************)
CASE iOUT_Step OF

(***** RESET *****)
ST100_Modify_e.RESET: (* Schritt 0-99 *)
    //Initialisierungen
    //Start Init Ablauf
    IF xIN_Init THEN
        iOUT_Step := ST100_Modify_e.INIT;
        //Start Manu Ablauf
    ELSIF enIN_State = StateMANU AND xIN_NextStep THEN
        iOUT_Step := ST100_Modify_e.INIT;
    END_IF;

(***** INIT *****)
ST100_Modify_e.INIT: (* Grundstellung ? *)
    IF TRUE THEN
        iOUT_Step := ST100_Modify_e.READY;
    ELSE
        iOUT_Step := ST100_Modify_e.INIT;
    END_IF;

(***** READY / INIT DONE *****)
ST100_Modify_e.READY: (* Start AUTO,END,LEER,STEP *)
    IF xIN_Start THEN //IF rtSTART.Q THEN
        iOUT_Step := ST100_Modify_e.START;
    END_IF

(***** START  ZYKLISCH *****)
ST100_Modify_e.START: (*  *)
    IF xIN_NextStep AND pxFG_Freigabe^ THEN
        iOUT_Step             := ST100_Modify_e.waitOnMover;
        iStartProcessTimeMili := GetTick();
    END_IF;

ST100_Modify_e.waitOnMover: (*  *)
    IF xIN_NextStep AND __ISVALIDREF(Mover) THEN
        iStartProcessTimeMili := GetTick();
        iOUT_Step             := ST100_Modify_e.proceedOperation_1;
    END_IF;

ST100_Modify_e.proceedOperation_1: (*  *)
    IF xIN_NextStep AND (GetTick() - iStartProcessTimeMili) >= (iProcessTimeMili1) THEN
        iStartProcessTimeMili := GetTick();
        iOUT_Step             := ST100_Modify_e.proceedOperation_2;
		_bBewegung := FALSE;
		
    ELSIF __ISVALIDREF(Mover) THEN
        IF Mover.MoverAxis.isInPos THEN
            IF _bBewegung THEN
                Mover.MoverAxis.RelMoveTo(_bBewegungDist);
            ELSE
                Mover.MoverAxis.RelMoveTo(-_bBewegungDist);
            END_IF

            _bBewegung := NOT _bBewegung;
        END_IF;
    END_IF;

ST100_Modify_e.proceedOperation_2: (*  *)
    IF xIN_NextStep AND (GetTick() - iStartProcessTimeMili) >= (iProcessTimeMili2) THEN
        iOUT_Step := ST100_Modify_e.SYNC_MOVER_LEAVE;
    END_IF;

ST100_Modify_e.SYNC_MOVER_LEAVE:
    // The mover needs to be taken by MoverMan
    IF NOT __ISVALIDREF(Mover) THEN
        iOUT_Step := ST100_Unload_e.DONE;
    END_IF

(***** DONE *****)
ST100_Modify_e.DONE: (* Letzter Schritt  *)
    IF NOT xIN_AlarmAktiv THEN
        //AUTO
        IF (enIN_State = StateAUTO) AND xIN_RestartCYCL THEN
            iOUT_Step := ST100_Modify_e.START;
            //STEP / END / LEERFAHREN restart
        ELSIF (enIN_State < StateAUTO) AND (enIN_State >= enState.StateSTEP) AND xIN_RestartCYCL THEN
            iOUT_Step := ST100_Modify_e.START;
            //STEP / END / LEERFAHREN fertig
        ELSIF (enIN_State = StateREADY) THEN
            iOUT_Step := ST100_Modify_e.READY;
        END_IF;
    END_IF;

(************ ERROR *************)
ST100_Modify_e.ERROR: (* ERROR *) ;

END_CASE;

END_FUNCTION_BLOCK

// ---- POUs/20_AUTO/ST180/FB_AUT_180.TcPOU
FUNCTION_BLOCK FB_AUT_180 EXTENDS FB_AUT_ABSTRACT
(****************************************************************************)
(*	POU_AUT_zxx			Bausteinaufrufe Station	zxx							*)
(*	Status				ungetestet											*)
(*  Version:			1.0													*)
(*	Beschrieb:																*)
(*																			*)
(*	Abläufe:			FB_ABLzxxA		Hauptablauf							*)
(*																			*)
(*																			*)
(* 	25.09.2019/Dj															*)
(****************************************************************************)
(*	dd.mm.yyyy   KZ    x.y			Beschrieb								*)
(****************************************************************************)
VAR_INPUT
    (* spezifische Eingänge *)

END_VAR
VAR_OUTPUT
    (* spezifische Ausgänge *)

END_VAR
VAR
    (* Bausteine *)
    fb_Pnp    : FB_ABL_180_Pnp;

    fb_stat : FB_AUT_Statistics;

END_VAR

(*******************************************************************)
(* Timer *)
(*******************************************************************)

(*******************************************************************)
(* Flanken / Merker *)
(*******************************************************************)
//MANU CYCLE
IF (enIN_State = StateMANU) AND xIN_ManuCycle THEN
    xManuCycle := TRUE;
END_IF;

IF (enIN_State <> StateMANU) OR xOUT_Done THEN
    xManuCycle := FALSE;
END_IF

//NEXT STEP
xNextStep := (enIN_State > StateSTEP) OR
             ((enIN_State = StateSTEP) AND xIN_Step) OR
             ((enIN_State = StateMANU) AND xManuCycle);

//RESET
xReset := (enIN_State < StateREADY) AND (enIN_State <> StateINIT) AND NOT xManuCycle;

(*******************************************************************)
(* Bausteinaufrufe Abläufe *)
(*******************************************************************)

xRelease := MAIN.MoverMan.IsProcessUsed(THIS^);

fb_Pnp(xIN_Reset          := xReset,
       xIN_Init           := xIN_Init,
       xIN_Quit           := xIN_Quit,
       xIN_Start          := enIN_State >= enState.StateLEER AND xRelease,
       xIN_Sperre         := NOT xIN_On,
       xIN_NextStep       := xNextStep,
       xIN_AlarmAktiv     := xIN_AlarmAktiv,
       xIN_DryCycle       := xIN_DryCycle,
       xIN_RestartCYCL    := enIN_State >= enState.StateLEER,
       enIN_State         := enIN_State,
       tIN_Timeout        := tIN_Timeout,
       pxFG_Freigabe      := ADR(xRelease),
       Mover              := THIS^.Mover,
       xIN_PceReadyToPick := TRUE);

